KUKA KRL program: EPS_2_251825_SA35_A_20260116064120.src

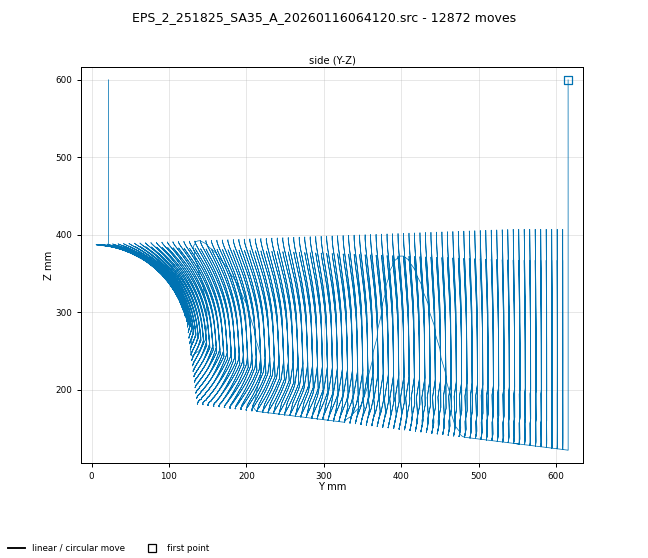
[picture p0: tool path of EPS_2_251825_SA35_A_20260116064120.src, 12872 of 12874 moves have a stored position in this frame; points joined in program order, loops and branches not executed]
&ACCESS RVP
&REL 4
&COMMENT QRS 19112012
&PARAM EDITMASK = *
DEF PART()
EXT BAS (BAS_COMMAND :IN,REAL :IN )
INT I
BAS (#INITMOV,0 )

;KUKA QRS Post kuka4.cps  Date:22-06-2017 !

File_ID=2990

QRS_PRE_INIT()

;Init var - Until changes are made in qrs_pre_init
Outlet_Square_prg=0
Inlet_1_Square_prg=0
Inlet_2_Square_prg=0
Inlet_3_Square_prg=0
Inlet_4_Square_prg=0
Inlet_5_Square_prg=0

Outlet_1={X 0.000, Y 546.330, Z 306.500, B 0.000, E1 0.000 }
Inlet_1={X 0.000, Y 549.180, Z 266.500, B 0.000, E1 180.000 }
Outlet_1_type=201
Inlet_1_type=201
;QRS#1=Sidecore dimensions
;QRS#2=200-8" PVC SDR 35
;QRS#3=200-8" PVC SDR 35
;QRS#4=
;QRS#5=
;QRS#6=
;QRS#7=
;QRS#8=
;QRS#9=12-08 PSX
;QRS#10=12-08 PSX
;QRS#11=
;QRS#12=
;QRS#13=
;QRS#14=
;QRS#15=
;QRS#16=1220x127x686 2,25'
;QRS#17=EPS Height
;QRS#18=407
;QRS#19=*
;QRS#20= UPDATED VERSION 22-06-2017
;QRS#21=*
Outlet_Square=0100
Inlet_1_Square=0100
Inlet_2_Square=0
Inlet_3_Square=0
Inlet_4_Square=0
Inlet_5_Square=0
Mill_Square=1
Outlet_Square_Prg=204
Inlet_1_Square_prg=204

QRS_INIT()

$ADVANCE=5

; T1
PTP {E1 173.649,E2 173.649}
PTP {X 0,Y 615.437,A -85,B 0,C 180,E1 173.649,E2 173.649,E3 0,E4 0,E5 0,E6 0}
QRS_SPEED_INIT()
LIN {X 0,Y 615.437,Z 600,A -85,B 0,C 180,E1 173.649,E2 173.649,E3 0,E4 0,E5 0,E6 0} C_VEL
LIN {X 0,Y 615.437,Z 131.876,A -85,B 0,C 180,E1 173.649,E2 173.649} C_VEL
LIN {X 0,Y 615.437,Z 123.698,A -85,B 0,C 180,E1 173.649,E2 173.649} C_VEL
LIN {X 0,Y 615.425,Z 121.698,A -85,B 0,C 180,E1 173.462,E2 173.462} C_VEL
LIN {X 0,Y 615.423,Z 121.698,A -85,B 0,C 180,E1 171.462,E2 171.462} C_VEL
LIN {X 0,Y 615.422,Z 121.699,A -85,B 0,C 180,E1 169.138,E2 169.138} C_VEL
LIN {X 0,Y 615.448,Z 121.699,A -85,B 0,C 180,E1 166.798,E2 166.798} C_VEL
LIN {X 0,Y 615.463,Z 121.696,A -85,B 0,C 180,E1 164.094,E2 164.094} C_VEL
LIN {X 0,Y 615.423,Z 121.698,A -85,B 0,C 180,E1 161.409,E2 161.409} C_VEL
LIN {X 0,Y 615.498,Z 121.698,A -85,B 0,C 180,E1 158.568,E2 158.568} C_VEL
LIN {X 0,Y 615.427,Z 121.697,A -85,B 0,C 180,E1 155.725,E2 155.725} C_VEL
LIN {X 0,Y 615.428,Z 121.697,A -85,B 0,C 180,E1 153.553,E2 153.553} C_VEL
LIN {X 0,Y 615.483,Z 121.695,A -85,B 0,C 180,E1 150.593,E2 150.593} C_VEL
LIN {X 0,Y 615.452,Z 121.694,A -85,B 0,C 180,E1 148.312,E2 148.312} C_VEL
LIN {X 0,Y 615.431,Z 121.696,A -85,B 0,C 180,E1 145.974,E2 145.974} C_VEL
LIN {X 0,Y 615.487,Z 121.703,A -85,B 0,C 180,E1 143.062,E2 143.062} C_VEL
LIN {X 0,Y 615.436,Z 121.695,A -85,B 0,C 180,E1 140.246,E2 140.246} C_VEL
LIN {X 0,Y 615.434,Z 121.697,A -85,B 0,C 180,E1 137.924,E2 137.924} C_VEL
LIN {X 0,Y 615.442,Z 121.697,A -85,B 0,C 180,E1 135.846,E2 135.846} C_VEL
LIN {X 0,Y 615.488,Z 121.693,A -85,B 0,C 180,E1 133.047,E2 133.047} C_VEL
LIN {X 0,Y 615.448,Z 121.693,A -85,B 0,C 180,E1 130.608,E2 130.608} C_VEL
LIN {X 0,Y 615.447,Z 121.697,A -85,B 0,C 180,E1 128.007,E2 128.007} C_VEL
LIN {X 0,Y 615.489,Z 121.7,A -85,B 0,C 180,E1 125.615,E2 125.615} C_VEL
LIN {X 0,Y 615.486,Z 121.691,A -85,B 0,C 180,E1 123.235,E2 123.235} C_VEL
LIN {X 0,Y 615.457,Z 121.691,A -85,B 0,C 180,E1 120.92,E2 120.92} C_VEL
LIN {X 0,Y 615.441,Z 121.695,A -85,B 0,C 180,E1 118.442,E2 118.442} C_VEL
LIN {X 0,Y 615.493,Z 121.693,A -85,B 0,C 180,E1 115.569,E2 115.569} C_VEL
LIN {X 0,Y 615.446,Z 121.692,A -85,B 0,C 180,E1 112.845,E2 112.845} C_VEL
LIN {X 0,Y 615.449,Z 121.695,A -85,B 0,C 180,E1 110.547,E2 110.547} C_VEL
LIN {X 0,Y 615.45,Z 121.868,A -85,B 0,C 180,E1 108.593,E2 108.593} C_VEL
LIN {X 0,Y 615.493,Z 137.711,A -85,B 0,C 180,E1 105.904,E2 105.904} C_VEL
LIN {X 0,Y 615.469,Z 154.863,A -85,B 0,C 180,E1 103.033,E2 103.033} C_VEL
LIN {X 0,Y 615.476,Z 156.121,A -85,B 0,C 180,E1 102.823,E2 102.823} C_VEL
LIN {X 0,Y 615.483,Z 263.822,A -85,B 0,C 180,E1 101.526,E2 101.526} C_VEL
LIN {X 0,Y 615.474,Z 276.761,A -85,B 0,C 180,E1 101.234,E2 101.234} C_VEL
LIN {X 0,Y 615.487,Z 288.668,A -85,B 0,C 180,E1 100.84,E2 100.84} C_VEL
LIN {X 0,Y 615.481,Z 301.206,A -85,B 0,C 180,E1 100.277,E2 100.277} C_VEL
LIN {X 0,Y 615.494,Z 312.583,A -85,B 0,C 180,E1 99.613,E2 99.613} C_VEL
LIN {X 0,Y 615.498,Z 322.829,A -85,B 0,C 180,E1 98.867,E2 98.867} C_VEL
LIN {X 0,Y 615.498,Z 332.038,A -85,B 0,C 180,E1 98.04,E2 98.04} C_VEL
LIN {X 0,Y 615.499,Z 340.895,A -85,B 0,C 180,E1 97.057,E2 97.057} C_VEL
LIN {X 0,Y 615.497,Z 348.126,A -85,B 0,C 180,E1 96.062,E2 96.062} C_VEL
LIN {X 0,Y 615.497,Z 352.96,A -85,B 0,C 180,E1 95.241,E2 95.241} C_VEL
LIN {X 0,Y 615.494,Z 357.66,A -85,B 0,C 180,E1 94.256,E2 94.256} C_VEL
LIN {X 0,Y 615.494,Z 361.256,A -85,B 0,C 180,E1 93.273,E2 93.273} C_VEL
LIN {X 0,Y 615.496,Z 363.116,A -85,B 0,C 180,E1 92.617,E2 92.617} C_VEL
LIN {X 0,Y 615.5,Z 364.533,A -85,B 0,C 180,E1 91.963,E2 91.963} C_VEL
LIN {X 0,Y 615.496,Z 366.142,A -85,B 0,C 180,E1 90.654,E2 90.654} C_VEL
LIN {X 0,Y 615.495,Z 366.384,A -85,B 0,C 180,E1 90,E2 90} C_VEL
LIN {X 0,Y 615.495,Z 366.205,A -85,B 0,C 180,E1 89.345,E2 89.345} C_VEL
LIN {X 0,Y 615.5,Z 364.682,A -85,B 0,C 180,E1 88.037,E2 88.037} C_VEL
LIN {X 0,Y 615.498,Z 363.341,A -85,B 0,C 180,E1 87.382,E2 87.382} C_VEL
LIN {X 0,Y 615.496,Z 360.493,A -85,B 0,C 180,E1 86.399,E2 86.399} C_VEL
LIN {X 0,Y 615.498,Z 356.633,A -85,B 0,C 180,E1 85.415,E2 85.415} C_VEL
LIN {X 0,Y 615.498,Z 351.65,A -85,B 0,C 180,E1 84.43,E2 84.43} C_VEL
LIN {X 0,Y 615.496,Z 345.208,A -85,B 0,C 180,E1 83.418,E2 83.418} C_VEL
LIN {X 0,Y 615.497,Z 337.535,A -85,B 0,C 180,E1 82.454,E2 82.454} C_VEL
LIN {X 0,Y 615.498,Z 327.756,A -85,B 0,C 180,E1 81.463,E2 81.463} C_VEL
LIN {X 0,Y 615.498,Z 317.49,A -85,B 0,C 180,E1 80.635,E2 80.635} C_VEL
LIN {X 0,Y 615.48,Z 305.928,A -85,B 0,C 180,E1 79.888,E2 79.888} C_VEL
LIN {X 0,Y 615.494,Z 294.071,A -85,B 0,C 180,E1 79.293,E2 79.293} C_VEL
LIN {X 0,Y 615.477,Z 281.156,A -85,B 0,C 180,E1 78.807,E2 78.807} C_VEL
LIN {X 0,Y 615.485,Z 268.552,A -85,B 0,C 180,E1 78.473,E2 78.473} C_VEL
LIN {X 0,Y 615.493,Z 255.419,A -85,B 0,C 180,E1 78.264,E2 78.264} C_VEL
LIN {X 0,Y 615.478,Z 156.153,A -85,B 0,C 180,E1 77.092,E2 77.092} C_VEL
LIN {X 0,Y 615.496,Z 139.253,A -85,B 0,C 180,E1 74.265,E2 74.265} C_VEL
LIN {X 0,Y 615.483,Z 124.248,A -85,B 0,C 180,E1 71.724,E2 71.724} C_VEL
LIN {X 0,Y 615.453,Z 121.694,A -85,B 0,C 180,E1 71.267,E2 71.267} C_VEL
LIN {X 0,Y 615.489,Z 121.686,A -85,B 0,C 180,E1 68.568,E2 68.568} C_VEL
LIN {X 0,Y 615.467,Z 121.697,A -85,B 0,C 180,E1 65.727,E2 65.727} C_VEL
LIN {X 0,Y 615.452,Z 121.695,A -85,B 0,C 180,E1 63.554,E2 63.554} C_VEL
LIN {X 0,Y 615.448,Z 121.692,A -85,B 0,C 180,E1 61.34,E2 61.34} C_VEL
LIN {X 0,Y 615.474,Z 121.688,A -85,B 0,C 180,E1 58.917,E2 58.917} C_VEL
LIN {X 0,Y 615.463,Z 121.697,A -85,B 0,C 180,E1 55.977,E2 55.977} C_VEL
LIN {X 0,Y 615.445,Z 121.693,A -85,B 0,C 180,E1 53.573,E2 53.573} C_VEL
LIN {X 0,Y 615.491,Z 121.688,A -85,B 0,C 180,E1 50.938,E2 50.938} C_VEL
LIN {X 0,Y 615.495,Z 121.701,A -85,B 0,C 180,E1 48.527,E2 48.527} C_VEL
LIN {X 0,Y 615.441,Z 121.694,A -85,B 0,C 180,E1 45.847,E2 45.847} C_VEL
LIN {X 0,Y 615.474,Z 121.69,A -85,B 0,C 180,E1 43.246,E2 43.246} C_VEL
LIN {X 0,Y 615.473,Z 121.7,A -85,B 0,C 180,E1 40.608,E2 40.608} C_VEL
LIN {X 0,Y 615.437,Z 121.696,A -85,B 0,C 180,E1 38.072,E2 38.072} C_VEL
LIN {X 0,Y 615.45,Z 121.693,A -85,B 0,C 180,E1 35.619,E2 35.619} C_VEL
LIN {X 0,Y 615.489,Z 121.694,A -85,B 0,C 180,E1 33.236,E2 33.236} C_VEL
LIN {X 0,Y 615.477,Z 121.701,A -85,B 0,C 180,E1 30.92,E2 30.92} C_VEL
LIN {X 0,Y 615.434,Z 121.697,A -85,B 0,C 180,E1 28.442,E2 28.442} C_VEL
LIN {X 0,Y 615.434,Z 121.697,A -85,B 0,C 180,E1 26.447,E2 26.447} C_VEL
LIN {X 0,Y 615.442,Z 121.694,A -85,B 0,C 180,E1 24,E2 24} C_VEL
LIN {X 0,Y 615.498,Z 121.696,A -85,B 0,C 180,E1 21.432,E2 21.432} C_VEL
LIN {X 0,Y 615.428,Z 121.697,A -85,B 0,C 180,E1 18.59,E2 18.59} C_VEL
LIN {X 0,Y 615.465,Z 121.695,A -85,B 0,C 180,E1 15.906,E2 15.906} C_VEL
LIN {X 0,Y 615.454,Z 121.699,A -85,B 0,C 180,E1 13.202,E2 13.202} C_VEL
LIN {X 0,Y 615.427,Z 121.698,A -85,B 0,C 180,E1 10.861,E2 10.861} C_VEL
LIN {X 0,Y 615.427,Z 121.697,A -85,B 0,C 180,E1 8.538,E2 8.538} C_VEL
LIN {X 0,Y 615.496,Z 121.696,A -85,B 0,C 180,E1 5.899,E2 5.899} C_VEL
LIN {X 0,Y 615.434,Z 121.699,A -85,B 0,C 180,E1 3.273,E2 3.273} C_VEL
LIN {X 0,Y 615.432,Z 121.699,A -85,B 0,C 180,E1 1.309,E2 1.309} C_VEL
LIN {X 0,Y 615.43,Z 121.699,A -85,B 0,C 180,E1 -0.654,E2 -0.654} C_VEL
LIN {X 0,Y 615.428,Z 121.699,A -85,B 0,C 180,E1 -2.618,E2 -2.618} C_VEL
LIN {X 0,Y 615.425,Z 121.7,A -85,B 0,C 180,E1 -4.585,E2 -4.585} C_VEL
LIN {X 0,Y 615.421,Z 121.7,A -85,B 0,C 180,E1 -6.557,E2 -6.557} C_VEL
LIN {X 0,Y 615.421,Z 121.7,A -85,B 0,C 180,E1 -8.538,E2 -8.538} C_VEL
LIN {X 0,Y 615.413,Z 121.7,A -85,B 0,C 180,E1 -10.855,E2 -10.855} C_VEL
LIN {X 0,Y 615.434,Z 121.7,A -85,B 0,C 180,E1 -13.202,E2 -13.202} C_VEL
LIN {X 0,Y 615.461,Z 121.699,A -85,B 0,C 180,E1 -15.906,E2 -15.906} C_VEL
LIN {X 0,Y 615.415,Z 121.7,A -85,B 0,C 180,E1 -18.648,E2 -18.648} C_VEL
LIN {X 0,Y 615.495,Z 121.7,A -85,B 0,C 180,E1 -21.432,E2 -21.432} C_VEL
LIN {X 0,Y 615.419,Z 121.699,A -85,B 0,C 180,E1 -24.275,E2 -24.275} C_VEL
LIN {X 0,Y 615.42,Z 121.699,A -85,B 0,C 180,E1 -26.447,E2 -26.447} C_VEL
LIN {X 0,Y 615.48,Z 121.698,A -85,B 0,C 180,E1 -29.407,E2 -29.407} C_VEL
LIN {X 0,Y 615.449,Z 121.696,A -85,B 0,C 180,E1 -31.688,E2 -31.688} C_VEL
LIN {X 0,Y 615.425,Z 121.697,A -85,B 0,C 180,E1 -34.026,E2 -34.026} C_VEL
LIN {X 0,Y 615.484,Z 121.7,A -85,B 0,C 180,E1 -36.937,E2 -36.937} C_VEL
LIN {X 0,Y 615.499,Z 121.697,A -85,B 0,C 180,E1 -39.064,E2 -39.064} C_VEL
LIN {X 0,Y 615.45,Z 121.695,A -85,B 0,C 180,E1 -41.477,E2 -41.477} C_VEL
LIN {X 0,Y 615.429,Z 121.697,A -85,B 0,C 180,E1 -43.992,E2 -43.992} C_VEL
LIN {X 0,Y 615.429,Z 121.697,A -85,B 0,C 180,E1 -46.008,E2 -46.008} C_VEL
LIN {X 0,Y 615.476,Z 121.699,A -85,B 0,C 180,E1 -48.526,E2 -48.526} C_VEL
LIN {X 0,Y 615.469,Z 121.693,A -85,B 0,C 180,E1 -51.095,E2 -51.095} C_VEL
LIN {X 0,Y 615.434,Z 121.695,A -85,B 0,C 180,E1 -53.572,E2 -53.572} C_VEL
LIN {X 0,Y 615.496,Z 121.701,A -85,B 0,C 180,E1 -56.465,E2 -56.465} C_VEL
LIN {X 0,Y 615.455,Z 121.692,A -85,B 0,C 180,E1 -59.079,E2 -59.079} C_VEL
LIN {X 0,Y 615.438,Z 121.695,A -85,B 0,C 180,E1 -61.559,E2 -61.559} C_VEL
LIN {X 0,Y 615.494,Z 121.695,A -85,B 0,C 180,E1 -64.43,E2 -64.43} C_VEL
LIN {X 0,Y 615.442,Z 121.693,A -85,B 0,C 180,E1 -67.154,E2 -67.154} C_VEL
LIN {X 0,Y 615.441,Z 121.788,A -85,B 0,C 180,E1 -67.44,E2 -67.44} C_VEL
LIN {X 0,Y 615.477,Z 140.398,A -85,B 0,C 180,E1 -69.967,E2 -69.967} C_VEL
LIN {X 0,Y 615.47,Z 161.077,A -85,B 0,C 180,E1 -72.729,E2 -72.729} C_VEL
LIN {X 0,Y 615.472,Z 181.732,A -85,B 0,C 180,E1 -75.45,E2 -75.45} C_VEL
LIN {X 0,Y 615.454,Z 194.469,A -85,B 0,C 180,E1 -77.113,E2 -77.113} C_VEL
LIN {X 0,Y 615.488,Z 302.82,A -85,B 0,C 180,E1 -78.41,E2 -78.41} C_VEL
LIN {X 0,Y 615.477,Z 315.339,A -85,B 0,C 180,E1 -78.681,E2 -78.681} C_VEL
LIN {X 0,Y 615.488,Z 328.617,A -85,B 0,C 180,E1 -79.113,E2 -79.113} C_VEL
LIN {X 0,Y 615.477,Z 340.475,A -85,B 0,C 180,E1 -79.639,E2 -79.639} C_VEL
LIN {X 0,Y 615.494,Z 351.991,A -85,B 0,C 180,E1 -80.304,E2 -80.304} C_VEL
LIN {X 0,Y 615.499,Z 362.338,A -85,B 0,C 180,E1 -81.05,E2 -81.05} C_VEL
LIN {X 0,Y 615.497,Z 370.809,A -85,B 0,C 180,E1 -81.794,E2 -81.794} C_VEL
LIN {X 0,Y 615.498,Z 378.604,A -85,B 0,C 180,E1 -82.619,E2 -82.619} C_VEL
LIN {X 0,Y 615.496,Z 386.201,A -85,B 0,C 180,E1 -83.608,E2 -83.608} C_VEL
LIN {X 0,Y 615.498,Z 393.203,A -85,B 0,C 180,E1 -84.759,E2 -84.759} C_VEL
LIN {X 0,Y 615.494,Z 397.85,A -85,B 0,C 180,E1 -85.743,E2 -85.743} C_VEL
LIN {X 0,Y 615.494,Z 401.398,A -85,B 0,C 180,E1 -86.727,E2 -86.727} C_VEL
LIN {X 0,Y 615.497,Z 403.232,A -85,B 0,C 180,E1 -87.382,E2 -87.382} C_VEL
LIN {X 0,Y 615.5,Z 404.607,A -85,B 0,C 180,E1 -88.037,E2 -88.037} C_VEL
LIN {X 0,Y 615.496,Z 406.173,A -85,B 0,C 180,E1 -89.345,E2 -89.345} C_VEL
LIN {X 0,Y 615.494,Z 406.389,A -85,B 0,C 180,E1 -90,E2 -90} C_VEL
LIN {X 0,Y 615.495,Z 405.58,A -85,B 0,C 180,E1 -91.308,E2 -91.308} C_VEL
LIN {X 0,Y 615.5,Z 404.608,A -85,B 0,C 180,E1 -91.963,E2 -91.963} C_VEL
LIN {X 0,Y 615.497,Z 403.234,A -85,B 0,C 180,E1 -92.617,E2 -92.617} C_VEL
LIN {X 0,Y 615.496,Z 400.351,A -85,B 0,C 180,E1 -93.6,E2 -93.6} C_VEL
LIN {X 0,Y 615.498,Z 396.443,A -85,B 0,C 180,E1 -94.584,E2 -94.584} C_VEL
LIN {X 0,Y 615.499,Z 391.407,A -85,B 0,C 180,E1 -95.569,E2 -95.569} C_VEL
LIN {X 0,Y 615.497,Z 384.869,A -85,B 0,C 180,E1 -96.583,E2 -96.583} C_VEL
LIN {X 0,Y 615.497,Z 377.137,A -85,B 0,C 180,E1 -97.545,E2 -97.545} C_VEL
LIN {X 0,Y 615.498,Z 369.05,A -85,B 0,C 180,E1 -98.371,E2 -98.371} C_VEL
LIN {X 0,Y 615.499,Z 359.174,A -85,B 0,C 180,E1 -99.198,E2 -99.198} C_VEL
LIN {X 0,Y 615.488,Z 347.99,A -85,B 0,C 180,E1 -99.945,E2 -99.945} C_VEL
LIN {X 0,Y 615.482,Z 337.034,A -85,B 0,C 180,E1 -100.527,E2 -100.527} C_VEL
LIN {X 0,Y 615.48,Z 324.497,A -85,B 0,C 180,E1 -101.04,E2 -101.04} C_VEL
LIN {X 0,Y 615.479,Z 312.09,A -85,B 0,C 180,E1 -101.401,E2 -101.401} C_VEL
LIN {X 0,Y 615.493,Z 298.502,A -85,B 0,C 180,E1 -101.651,E2 -101.651} C_VEL
LIN {X 0,Y 615.454,Z 194.475,A -85,B 0,C 180,E1 -102.887,E2 -102.887} C_VEL
LIN {X 0,Y 615.496,Z 172.701,A -85,B 0,C 180,E1 -105.734,E2 -105.734} C_VEL
LIN {X 0,Y 615.455,Z 152.32,A -85,B 0,C 180,E1 -108.436,E2 -108.436} C_VEL
LIN {X 0,Y 615.475,Z 132.642,A -85,B 0,C 180,E1 -111.081,E2 -111.081} C_VEL
LIN {X 0,Y 615.44,Z 121.695,A -85,B 0,C 180,E1 -112.591,E2 -112.591} C_VEL
LIN {X 0,Y 615.452,Z 121.692,A -85,B 0,C 180,E1 -114.993,E2 -114.993} C_VEL
LIN {X 0,Y 615.472,Z 121.699,A -85,B 0,C 180,E1 -117.915,E2 -117.915} C_VEL
LIN {X 0,Y 615.446,Z 121.697,A -85,B 0,C 180,E1 -120.161,E2 -120.161} C_VEL
LIN {X 0,Y 615.436,Z 121.695,A -85,B 0,C 180,E1 -122.46,E2 -122.46} C_VEL
LIN {X 0,Y 615.453,Z 121.693,A -85,B 0,C 180,E1 -124.816,E2 -124.816} C_VEL
LIN {X 0,Y 615.498,Z 121.694,A -85,B 0,C 180,E1 -127.24,E2 -127.24} C_VEL
LIN {X 0,Y 615.454,Z 121.698,A -85,B 0,C 180,E1 -129.752,E2 -129.752} C_VEL
LIN {X 0,Y 615.431,Z 121.697,A -85,B 0,C 180,E1 -132.074,E2 -132.074} C_VEL
LIN {X 0,Y 615.43,Z 121.696,A -85,B 0,C 180,E1 -134.153,E2 -134.153} C_VEL
LIN {X 0,Y 615.471,Z 121.693,A -85,B 0,C 180,E1 -136.754,E2 -136.754} C_VEL
LIN {X 0,Y 615.457,Z 121.7,A -85,B 0,C 180,E1 -139.391,E2 -139.391} C_VEL
LIN {X 0,Y 615.493,Z 121.7,A -85,B 0,C 180,E1 -141.096,E2 -141.096} C_VEL
LIN {X 0,Y 615.432,Z 121.699,A -85,B 0,C 180,E1 -143.571,E2 -143.571} C_VEL
LIN {X 0,Y 615.427,Z 121.697,A -85,B 0,C 180,E1 -145.974,E2 -145.974} C_VEL
LIN {X 0,Y 615.482,Z 121.701,A -85,B 0,C 180,E1 -148.913,E2 -148.913} C_VEL
LIN {X 0,Y 615.424,Z 121.698,A -85,B 0,C 180,E1 -151.558,E2 -151.558} C_VEL
LIN {X 0,Y 615.422,Z 121.698,A -85,B 0,C 180,E1 -153.553,E2 -153.553} C_VEL
LIN {X 0,Y 615.436,Z 121.697,A -85,B 0,C 180,E1 -156,E2 -156} C_VEL
LIN {X 0,Y 615.498,Z 121.7,A -85,B 0,C 180,E1 -158.568,E2 -158.568} C_VEL
LIN {X 0,Y 615.415,Z 121.7,A -85,B 0,C 180,E1 -161.412,E2 -161.412} C_VEL
LIN {X 0,Y 615.462,Z 121.698,A -85,B 0,C 180,E1 -164.094,E2 -164.094} C_VEL
LIN {X 0,Y 615.439,Z 121.7,A -85,B 0,C 180,E1 -166.798,E2 -166.798} C_VEL
LIN {X 0,Y 615.415,Z 121.7,A -85,B 0,C 180,E1 -169.141,E2 -169.141} C_VEL
LIN {X 0,Y 615.419,Z 121.7,A -85,B 0,C 180,E1 -171.462,E2 -171.462} C_VEL
LIN {X 0,Y 615.496,Z 121.7,A -85,B 0,C 180,E1 -174.102,E2 -174.102} C_VEL
LIN {X 0,Y 615.422,Z 121.7,A -85,B 0,C 180,E1 -176.727,E2 -176.727} C_VEL
LIN {X 0,Y 615.422,Z 121.7,A -85,B 0,C 180,E1 -178.691,E2 -178.691} C_VEL
LIN {X 0,Y 615.423,Z 121.699,A -85,B 0,C 180,E1 -180.654,E2 -180.654} C_VEL
LIN {X 0,Y 615.424,Z 121.699,A -85,B 0,C 180,E1 -182.618,E2 -182.618} C_VEL
LIN {X 0,Y 615.424,Z 121.699,A -85,B 0,C 180,E1 -184.585,E2 -184.585} C_VEL
LIN {X 0,Y 615.425,Z 121.698,A -85,B 0,C 180,E1 -186.538,E2 -186.538} C_VEL
LIN {X 0,Y 614.752,Z 121.846,A -85,B 0,C 180,E1 -187.084,E2 -187.084} C_VEL
LIN {X 0,Y 611.92,Z 122.262,A -85,B 0,C 180,E1 -187.97,E2 -187.97} C_VEL
LIN {X 0,Y 609.535,Z 122.57,A -85,B 0,C 180,E1 -188.683,E2 -188.683} C_VEL
LIN {X 0,Y 608.512,Z 122.685,A -85,B 0,C 180,E1 -189.233,E2 -189.233} C_VEL
LIN {X 0,Y 608.428,Z 122.694,A -85,B 0,C 180,E1 -189.419,E2 -189.419} C_VEL
LIN {X 0,Y 608.441,Z 122.693,A -85,B 0,C 180,E1 -192,E2 -192} C_VEL
LIN {X 0,Y 608.394,Z 122.695,A -85,B 0,C 180,E1 -194.723,E2 -194.723} C_VEL
LIN {X 0,Y 608.431,Z 122.701,A -85,B 0,C 180,E1 -197.477,E2 -197.477} C_VEL
LIN {X 0,Y 608.413,Z 122.693,A -85,B 0,C 180,E1 -200.276,E2 -200.276} C_VEL
LIN {X 0,Y 608.419,Z 122.692,A -85,B 0,C 180,E1 -202.47,E2 -202.47} C_VEL
LIN {X 0,Y 608.436,Z 122.7,A -85,B 0,C 180,E1 -205.302,E2 -205.302} C_VEL
LIN {X 0,Y 608.429,Z 122.696,A -85,B 0,C 180,E1 -207.519,E2 -207.519} C_VEL
LIN {X 0,Y 608.408,Z 122.693,A -85,B 0,C 180,E1 -209.964,E2 -209.964} C_VEL
LIN {X 0,Y 608.42,Z 122.694,A -85,B 0,C 180,E1 -212.518,E2 -212.518} C_VEL
LIN {X 0,Y 608.419,Z 122.697,A -85,B 0,C 180,E1 -215.279,E2 -215.279} C_VEL
LIN {X 0,Y 608.435,Z 122.69,A -85,B 0,C 180,E1 -217.749,E2 -217.749} C_VEL
LIN {X 0,Y 608.426,Z 122.693,A -85,B 0,C 180,E1 -220.328,E2 -220.328} C_VEL
LIN {X 0,Y 608.46,Z 122.689,A -85,B 0,C 180,E1 -223.309,E2 -223.309} C_VEL
LIN {X 0,Y 608.434,Z 122.692,A -85,B 0,C 180,E1 -226.129,E2 -226.129} C_VEL
LIN {X 0,Y 608.457,Z 122.694,A -85,B 0,C 180,E1 -228.825,E2 -228.825} C_VEL
LIN {X 0,Y 608.435,Z 122.69,A -85,B 0,C 180,E1 -231.764,E2 -231.764} C_VEL
LIN {X 0,Y 608.433,Z 122.693,A -85,B 0,C 180,E1 -233.957,E2 -233.957} C_VEL
LIN {X 0,Y 608.464,Z 122.696,A -85,B 0,C 180,E1 -236.33,E2 -236.33} C_VEL
LIN {X 0,Y 608.443,Z 122.693,A -85,B 0,C 180,E1 -238.734,E2 -238.734} C_VEL
LIN {X 0,Y 608.435,Z 122.69,A -85,B 0,C 180,E1 -241.387,E2 -241.387} C_VEL
LIN {X 0,Y 608.433,Z 122.697,A -85,B 0,C 180,E1 -243.965,E2 -243.965} C_VEL
LIN {X 0,Y 608.432,Z 122.691,A -85,B 0,C 180,E1 -246.876,E2 -246.876} C_VEL
LIN {X 0,Y 608.438,Z 122.691,A -85,B 0,C 180,E1 -249.33,E2 -249.33} C_VEL
LIN {X 0,Y 608.462,Z 122.864,A -85,B 0,C 180,E1 -251.345,E2 -251.345} C_VEL
LIN {X 0,Y 608.499,Z 138.846,A -85,B 0,C 180,E1 -254.08,E2 -254.08} C_VEL
LIN {X 0,Y 608.448,Z 155.056,A -85,B 0,C 180,E1 -256.814,E2 -256.814} C_VEL
LIN {X 0,Y 608.464,Z 156.323,A -85,B 0,C 180,E1 -257.026,E2 -257.026} C_VEL
LIN {X 0,Y 608.56,Z 165.703,A -85,B 0,C 180,E1 -257.156,E2 -257.156} C_VEL
LIN {X 0,Y 608.554,Z 262.824,A -85,B 0,C 180,E1 -258.32,E2 -258.32} C_VEL
LIN {X 0,Y 608.524,Z 276.133,A -85,B 0,C 180,E1 -258.614,E2 -258.614} C_VEL
LIN {X 0,Y 608.522,Z 289.437,A -85,B 0,C 180,E1 -259.058,E2 -259.058} C_VEL
LIN {X 0,Y 608.494,Z 301.378,A -85,B 0,C 180,E1 -259.604,E2 -259.604} C_VEL
LIN {X 0,Y 608.506,Z 312.797,A -85,B 0,C 180,E1 -260.276,E2 -260.276} C_VEL
LIN {X 0,Y 608.474,Z 323.09,A -85,B 0,C 180,E1 -261.03,E2 -261.03} C_VEL
LIN {X 0,Y 608.464,Z 332.354,A -85,B 0,C 180,E1 -261.866,E2 -261.866} C_VEL
LIN {X 0,Y 608.466,Z 341.327,A -85,B 0,C 180,E1 -262.868,E2 -262.868} C_VEL
LIN {X 0,Y 608.444,Z 348.558,A -85,B 0,C 180,E1 -263.867,E2 -263.867} C_VEL
LIN {X 0,Y 608.462,Z 353.437,A -85,B 0,C 180,E1 -264.699,E2 -264.699} C_VEL
LIN {X 0,Y 608.439,Z 358.18,A -85,B 0,C 180,E1 -265.695,E2 -265.695} C_VEL
LIN {X 0,Y 608.425,Z 361.813,A -85,B 0,C 180,E1 -266.689,E2 -266.689} C_VEL
LIN {X 0,Y 608.425,Z 363.692,A -85,B 0,C 180,E1 -267.352,E2 -267.352} C_VEL
LIN {X 0,Y 608.445,Z 365.127,A -85,B 0,C 180,E1 -268.015,E2 -268.015} C_VEL
LIN {X 0,Y 608.439,Z 366.752,A -85,B 0,C 180,E1 -269.339,E2 -269.339} C_VEL
LIN {X 0,Y 608.435,Z 366.996,A -85,B 0,C 180,E1 -270,E2 -270} C_VEL
LIN {X 0,Y 608.438,Z 366.815,A -85,B 0,C 180,E1 -270.662,E2 -270.662} C_VEL
LIN {X 0,Y 608.445,Z 365.276,A -85,B 0,C 180,E1 -271.986,E2 -271.986} C_VEL
LIN {X 0,Y 608.426,Z 363.918,A -85,B 0,C 180,E1 -272.649,E2 -272.649} C_VEL
LIN {X 0,Y 608.449,Z 361.041,A -85,B 0,C 180,E1 -273.643,E2 -273.643} C_VEL
LIN {X 0,Y 608.433,Z 357.142,A -85,B 0,C 180,E1 -274.638,E2 -274.638} C_VEL
LIN {X 0,Y 608.45,Z 352.111,A -85,B 0,C 180,E1 -275.635,E2 -275.635} C_VEL
LIN {X 0,Y 608.441,Z 345.793,A -85,B 0,C 180,E1 -276.633,E2 -276.633} C_VEL
LIN {X 0,Y 608.475,Z 337.876,A -85,B 0,C 180,E1 -277.633,E2 -277.633} C_VEL
LIN {X 0,Y 608.472,Z 328.034,A -85,B 0,C 180,E1 -278.636,E2 -278.636} C_VEL
LIN {X 0,Y 608.48,Z 317.711,A -85,B 0,C 180,E1 -279.474,E2 -279.474} C_VEL
LIN {X 0,Y 608.476,Z 306.096,A -85,B 0,C 180,E1 -280.229,E2 -280.229} C_VEL
LIN {X 0,Y 608.51,Z 294.204,A -85,B 0,C 180,E1 -280.831,E2 -280.831} C_VEL
LIN {X 0,Y 608.52,Z 281.256,A -85,B 0,C 180,E1 -281.323,E2 -281.323} C_VEL
LIN {X 0,Y 608.544,Z 268.637,A -85,B 0,C 180,E1 -281.66,E2 -281.66} C_VEL
LIN {X 0,Y 608.556,Z 255.527,A -85,B 0,C 180,E1 -281.871,E2 -281.871} C_VEL
LIN {X 0,Y 608.45,Z 156.349,A -85,B 0,C 180,E1 -283.059,E2 -283.059} C_VEL
LIN {X 0,Y 608.497,Z 139.372,A -85,B 0,C 180,E1 -285.921,E2 -285.921} C_VEL
LIN {X 0,Y 608.47,Z 122.894,A -85,B 0,C 180,E1 -288.739,E2 -288.739} C_VEL
LIN {X 0,Y 608.441,Z 122.689,A -85,B 0,C 180,E1 -290.982,E2 -290.982} C_VEL
LIN {X 0,Y 608.469,Z 122.694,A -85,B 0,C 180,E1 -293.845,E2 -293.845} C_VEL
LIN {X 0,Y 608.436,Z 122.698,A -85,B 0,C 180,E1 -296.036,E2 -296.036} C_VEL
LIN {X 0,Y 608.442,Z 122.689,A -85,B 0,C 180,E1 -298.614,E2 -298.614} C_VEL
LIN {X 0,Y 608.446,Z 122.691,A -85,B 0,C 180,E1 -301.267,E2 -301.267} C_VEL
LIN {X 0,Y 608.474,Z 122.695,A -85,B 0,C 180,E1 -303.735,E2 -303.735} C_VEL
LIN {X 0,Y 608.437,Z 122.692,A -85,B 0,C 180,E1 -306.093,E2 -306.093} C_VEL
LIN {X 0,Y 608.421,Z 122.692,A -85,B 0,C 180,E1 -308.591,E2 -308.591} C_VEL
LIN {X 0,Y 608.468,Z 122.694,A -85,B 0,C 180,E1 -311.342,E2 -311.342} C_VEL
LIN {X 0,Y 608.44,Z 122.692,A -85,B 0,C 180,E1 -313.872,E2 -313.872} C_VEL
LIN {X 0,Y 608.462,Z 122.688,A -85,B 0,C 180,E1 -316.692,E2 -316.692} C_VEL
LIN {X 0,Y 608.431,Z 122.694,A -85,B 0,C 180,E1 -319.673,E2 -319.673} C_VEL
LIN {X 0,Y 608.439,Z 122.689,A -85,B 0,C 180,E1 -322.251,E2 -322.251} C_VEL
LIN {X 0,Y 608.445,Z 122.699,A -85,B 0,C 180,E1 -325.095,E2 -325.095} C_VEL
LIN {X 0,Y 608.426,Z 122.691,A -85,B 0,C 180,E1 -327.903,E2 -327.903} C_VEL
LIN {X 0,Y 608.435,Z 122.691,A -85,B 0,C 180,E1 -330.219,E2 -330.219} C_VEL
LIN {X 0,Y 608.481,Z 122.694,A -85,B 0,C 180,E1 -332.791,E2 -332.791} C_VEL
LIN {X 0,Y 608.421,Z 122.693,A -85,B 0,C 180,E1 -335.427,E2 -335.427} C_VEL
LIN {X 0,Y 608.457,Z 122.691,A -85,B 0,C 180,E1 -338.308,E2 -338.308} C_VEL
LIN {X 0,Y 608.413,Z 122.694,A -85,B 0,C 180,E1 -341.299,E2 -341.299} C_VEL
LIN {X 0,Y 608.427,Z 122.692,A -85,B 0,C 180,E1 -343.905,E2 -343.905} C_VEL
LIN {X 0,Y 608.438,Z 122.697,A -85,B 0,C 180,E1 -346.643,E2 -346.643} C_VEL
LIN {X 0,Y 608.408,Z 122.693,A -85,B 0,C 180,E1 -349.349,E2 -349.349} C_VEL
LIN {X 0,Y 608.467,Z 122.692,A -85,B 0,C 180,E1 -352.033,E2 -352.033} C_VEL
LIN {X 0,Y 608.424,Z 122.694,A -85,B 0,C 180,E1 -354.698,E2 -354.698} C_VEL
LIN {X 0,Y 608.422,Z 122.692,A -85,B 0,C 180,E1 -357.352,E2 -357.352} C_VEL
LIN {X 0,Y 608.471,Z 122.695,A -85,B 0,C 180,E1 -360,E2 -360} C_VEL
LIN {X 0,Y 608.424,Z 122.693,A -85,B 0,C 180,E1 -362.648,E2 -362.648} C_VEL
LIN {X 0,Y 608.412,Z 122.694,A -85,B 0,C 180,E1 -365.302,E2 -365.302} C_VEL
LIN {X 0,Y 608.461,Z 122.695,A -85,B 0,C 180,E1 -367.967,E2 -367.967} C_VEL
LIN {X 0,Y 608.398,Z 122.695,A -85,B 0,C 180,E1 -370.651,E2 -370.651} C_VEL
LIN {X 0,Y 608.423,Z 122.696,A -85,B 0,C 180,E1 -373.357,E2 -373.357} C_VEL
LIN {X 0,Y 608.421,Z 122.695,A -85,B 0,C 180,E1 -376.095,E2 -376.095} C_VEL
LIN {X 0,Y 608.422,Z 122.693,A -85,B 0,C 180,E1 -378.871,E2 -378.871} C_VEL
LIN {X 0,Y 608.452,Z 122.694,A -85,B 0,C 180,E1 -381.692,E2 -381.692} C_VEL
LIN {X 0,Y 608.406,Z 122.694,A -85,B 0,C 180,E1 -384.573,E2 -384.573} C_VEL
LIN {X 0,Y 608.467,Z 122.695,A -85,B 0,C 180,E1 -387.206,E2 -387.206} C_VEL
LIN {X 0,Y 608.404,Z 122.694,A -85,B 0,C 180,E1 -389.962,E2 -389.962} C_VEL
LIN {X 0,Y 608.413,Z 122.694,A -85,B 0,C 180,E1 -392.516,E2 -392.516} C_VEL
LIN {X 0,Y 608.413,Z 122.699,A -85,B 0,C 180,E1 -395.28,E2 -395.28} C_VEL
LIN {X 0,Y 608.431,Z 122.691,A -85,B 0,C 180,E1 -397.749,E2 -397.749} C_VEL
LIN {X 0,Y 608.431,Z 122.692,A -85,B 0,C 180,E1 -400.327,E2 -400.327} C_VEL
LIN {X 0,Y 608.459,Z 122.69,A -85,B 0,C 180,E1 -403.308,E2 -403.308} C_VEL
LIN {X 0,Y 608.427,Z 122.692,A -85,B 0,C 180,E1 -406.127,E2 -406.127} C_VEL
LIN {X 0,Y 608.455,Z 122.695,A -85,B 0,C 180,E1 -408.824,E2 -408.824} C_VEL
LIN {X 0,Y 608.412,Z 122.693,A -85,B 0,C 180,E1 -411.408,E2 -411.408} C_VEL
LIN {X 0,Y 608.43,Z 122.692,A -85,B 0,C 180,E1 -413.907,E2 -413.907} C_VEL
LIN {X 0,Y 608.447,Z 122.696,A -85,B 0,C 180,E1 -416.328,E2 -416.328} C_VEL
LIN {X 0,Y 608.444,Z 122.694,A -85,B 0,C 180,E1 -418.733,E2 -418.733} C_VEL
LIN {X 0,Y 608.433,Z 122.69,A -85,B 0,C 180,E1 -421.387,E2 -421.387} C_VEL
LIN {X 0,Y 608.43,Z 122.696,A -85,B 0,C 180,E1 -423.964,E2 -423.964} C_VEL
LIN {X 0,Y 608.43,Z 122.693,A -85,B 0,C 180,E1 -426.875,E2 -426.875} C_VEL
LIN {X 0,Y 608.435,Z 122.82,A -85,B 0,C 180,E1 -427.309,E2 -427.309} C_VEL
LIN {X 0,Y 608.573,Z 138.08,A -85,B 0,C 180,E1 -429.412,E2 -429.412} C_VEL
LIN {X 0,Y 608.532,Z 158.529,A -85,B 0,C 180,E1 -432.179,E2 -432.179} C_VEL
LIN {X 0,Y 608.493,Z 179.24,A -85,B 0,C 180,E1 -434.937,E2 -434.937} C_VEL
LIN {X 0,Y 608.441,Z 194.612,A -85,B 0,C 180,E1 -436.962,E2 -436.962} C_VEL
LIN {X 0,Y 608.564,Z 247,A -85,B 0,C 180,E1 -437.6,E2 -437.6} C_VEL
LIN {X 0,Y 608.547,Z 302.937,A -85,B 0,C 180,E1 -438.276,E2 -438.276} C_VEL
LIN {X 0,Y 608.512,Z 316.21,A -85,B 0,C 180,E1 -438.571,E2 -438.571} C_VEL
LIN {X 0,Y 608.514,Z 328.627,A -85,B 0,C 180,E1 -438.982,E2 -438.982} C_VEL
LIN {X 0,Y 608.499,Z 340.631,A -85,B 0,C 180,E1 -439.519,E2 -439.519} C_VEL
LIN {X 0,Y 608.484,Z 352.194,A -85,B 0,C 180,E1 -440.191,E2 -440.191} C_VEL
LIN {X 0,Y 608.485,Z 362.591,A -85,B 0,C 180,E1 -440.946,E2 -440.946} C_VEL
LIN {X 0,Y 608.475,Z 371.109,A -85,B 0,C 180,E1 -441.699,E2 -441.699} C_VEL
LIN {X 0,Y 608.471,Z 378.958,A -85,B 0,C 180,E1 -442.534,E2 -442.534} C_VEL
LIN {X 0,Y 608.461,Z 386.286,A -85,B 0,C 180,E1 -443.484,E2 -443.484} C_VEL
LIN {X 0,Y 608.451,Z 391.864,A -85,B 0,C 180,E1 -444.365,E2 -444.365} C_VEL
LIN {X 0,Y 608.432,Z 396.949,A -85,B 0,C 180,E1 -445.362,E2 -445.362} C_VEL
LIN {X 0,Y 608.449,Z 400.895,A -85,B 0,C 180,E1 -446.357,E2 -446.357} C_VEL
LIN {X 0,Y 608.425,Z 403.808,A -85,B 0,C 180,E1 -447.351,E2 -447.351} C_VEL
LIN {X 0,Y 608.445,Z 405.201,A -85,B 0,C 180,E1 -448.014,E2 -448.014} C_VEL
LIN {X 0,Y 608.438,Z 406.783,A -85,B 0,C 180,E1 -449.338,E2 -449.338} C_VEL
LIN {X 0,Y 608.434,Z 407,A -85,B 0,C 180,E1 -450,E2 -450} C_VEL
LIN {X 0,Y 608.448,Z 406.184,A -85,B 0,C 180,E1 -451.323,E2 -451.323} C_VEL
LIN {X 0,Y 608.445,Z 405.202,A -85,B 0,C 180,E1 -451.985,E2 -451.985} C_VEL
LIN {X 0,Y 608.425,Z 403.81,A -85,B 0,C 180,E1 -452.648,E2 -452.648} C_VEL
LIN {X 0,Y 608.449,Z 400.897,A -85,B 0,C 180,E1 -453.642,E2 -453.642} C_VEL
LIN {X 0,Y 608.432,Z 396.952,A -85,B 0,C 180,E1 -454.637,E2 -454.637} C_VEL
LIN {X 0,Y 608.438,Z 390.879,A -85,B 0,C 180,E1 -455.8,E2 -455.8} C_VEL
LIN {X 0,Y 608.462,Z 384.238,A -85,B 0,C 180,E1 -456.799,E2 -456.799} C_VEL
LIN {X 0,Y 608.456,Z 375.993,A -85,B 0,C 180,E1 -457.8,E2 -457.8} C_VEL
LIN {X 0,Y 608.472,Z 367.542,A -85,B 0,C 180,E1 -458.635,E2 -458.635} C_VEL
LIN {X 0,Y 608.479,Z 357.098,A -85,B 0,C 180,E1 -459.473,E2 -459.473} C_VEL
LIN {X 0,Y 608.489,Z 346.764,A -85,B 0,C 180,E1 -460.144,E2 -460.144} C_VEL
LIN {X 0,Y 608.519,Z 335.275,A -85,B 0,C 180,E1 -460.74,E2 -460.74} C_VEL
LIN {X 0,Y 608.528,Z 322.903,A -85,B 0,C 180,E1 -461.224,E2 -461.224} C_VEL
LIN {X 0,Y 608.544,Z 309.461,A -85,B 0,C 180,E1 -461.596,E2 -461.596} C_VEL
LIN {X 0,Y 608.553,Z 297.125,A -85,B 0,C 180,E1 -461.807,E2 -461.807} C_VEL
LIN {X 0,Y 608.496,Z 195.189,A -85,B 0,C 180,E1 -463.015,E2 -463.015} C_VEL
LIN {X 0,Y 608.444,Z 194.132,A -85,B 0,C 180,E1 -463.101,E2 -463.101} C_VEL
LIN {X 0,Y 608.497,Z 172.773,A -85,B 0,C 180,E1 -465.92,E2 -465.92} C_VEL
LIN {X 0,Y 608.498,Z 151.84,A -85,B 0,C 180,E1 -468.723,E2 -468.723} C_VEL
LIN {X 0,Y 608.574,Z 131.351,A -85,B 0,C 180,E1 -471.509,E2 -471.509} C_VEL
LIN {X 0,Y 608.424,Z 122.693,A -85,B 0,C 180,E1 -472.715,E2 -472.715} C_VEL
LIN {X 0,Y 608.438,Z 122.693,A -85,B 0,C 180,E1 -475.301,E2 -475.301} C_VEL
LIN {X 0,Y 608.437,Z 122.697,A -85,B 0,C 180,E1 -477.518,E2 -477.518} C_VEL
LIN {X 0,Y 608.433,Z 122.695,A -85,B 0,C 180,E1 -479.965,E2 -479.965} C_VEL
LIN {X 0,Y 608.419,Z 122.692,A -85,B 0,C 180,E1 -482.516,E2 -482.516} C_VEL
LIN {X 0,Y 608.422,Z 122.693,A -85,B 0,C 180,E1 -484.901,E2 -484.901} C_VEL
LIN {X 0,Y 608.442,Z 122.694,A -85,B 0,C 180,E1 -487.747,E2 -487.747} C_VEL
LIN {X 0,Y 608.427,Z 122.691,A -85,B 0,C 180,E1 -490.326,E2 -490.326} C_VEL
LIN {X 0,Y 608.481,Z 122.694,A -85,B 0,C 180,E1 -493.31,E2 -493.31} C_VEL
LIN {X 0,Y 608.425,Z 122.691,A -85,B 0,C 180,E1 -496.126,E2 -496.126} C_VEL
LIN {X 0,Y 608.448,Z 122.694,A -85,B 0,C 180,E1 -498.823,E2 -498.823} C_VEL
LIN {X 0,Y 608.424,Z 122.692,A -85,B 0,C 180,E1 -501.763,E2 -501.763} C_VEL
LIN {X 0,Y 608.42,Z 122.692,A -85,B 0,C 180,E1 -503.956,E2 -503.956} C_VEL
LIN {X 0,Y 608.434,Z 122.692,A -85,B 0,C 180,E1 -506.327,E2 -506.327} C_VEL
LIN {X 0,Y 608.438,Z 122.698,A -85,B 0,C 180,E1 -508.732,E2 -508.732} C_VEL
LIN {X 0,Y 608.424,Z 122.693,A -85,B 0,C 180,E1 -511.386,E2 -511.386} C_VEL
LIN {X 0,Y 608.409,Z 122.696,A -85,B 0,C 180,E1 -513.224,E2 -513.224} C_VEL
LIN {X 0,Y 608.407,Z 122.694,A -85,B 0,C 180,E1 -515.86,E2 -515.86} C_VEL
LIN {X 0,Y 608.454,Z 122.693,A -85,B 0,C 180,E1 -518.308,E2 -518.308} C_VEL
LIN {X 0,Y 608.402,Z 122.694,A -85,B 0,C 180,E1 -521.3,E2 -521.3} C_VEL
LIN {X 0,Y 608.422,Z 122.694,A -85,B 0,C 180,E1 -523.905,E2 -523.905} C_VEL
LIN {X 0,Y 608.426,Z 122.696,A -85,B 0,C 180,E1 -526.643,E2 -526.643} C_VEL
LIN {X 0,Y 608.399,Z 122.694,A -85,B 0,C 180,E1 -529.349,E2 -529.349} C_VEL
LIN {X 0,Y 608.458,Z 122.695,A -85,B 0,C 180,E1 -532.033,E2 -532.033} C_VEL
LIN {X 0,Y 608.412,Z 122.695,A -85,B 0,C 180,E1 -534.698,E2 -534.698} C_VEL
LIN {X 0,Y 608.416,Z 122.693,A -85,B 0,C 180,E1 -537.352,E2 -537.352} C_VEL
LIN {X 0,Y 608.466,Z 122.696,A -85,B 0,C 180,E1 -540,E2 -540} C_VEL
LIN {X 0,Y 608.419,Z 122.692,A -85,B 0,C 180,E1 -542.648,E2 -542.648} C_VEL
LIN {X 0,Y 608.418,Z 122.694,A -85,B 0,C 180,E1 -545.302,E2 -545.302} C_VEL
LIN {X 0,Y 608.463,Z 122.693,A -85,B 0,C 180,E1 -547.967,E2 -547.967} C_VEL
LIN {X 0,Y 608.428,Z 122.694,A -85,B 0,C 180,E1 -549.419,E2 -549.419} C_VEL
LIN {X 0,Y 607.765,Z 122.779,A -85,B 0,C 180,E1 -549.971,E2 -549.971} C_VEL
LIN {X 0,Y 604.926,Z 123.131,A -85,B 0,C 180,E1 -550.868,E2 -550.868} C_VEL
LIN {X 0,Y 602.515,Z 123.437,A -85,B 0,C 180,E1 -551.589,E2 -551.589} C_VEL
LIN {X 0,Y 601.463,Z 123.561,A -85,B 0,C 180,E1 -552.146,E2 -552.146} C_VEL
LIN {X 0,Y 601.369,Z 123.571,A -85,B 0,C 180,E1 -552.334,E2 -552.334} C_VEL
LIN {X 0,Y 601.371,Z 123.571,A -85,B 0,C 180,E1 -554.899,E2 -554.899} C_VEL
LIN {X 0,Y 601.37,Z 123.577,A -85,B 0,C 180,E1 -557.689,E2 -557.689} C_VEL
LIN {X 0,Y 601.378,Z 123.573,A -85,B 0,C 180,E1 -559.81,E2 -559.81} C_VEL
LIN {X 0,Y 601.39,Z 123.569,A -85,B 0,C 180,E1 -562.684,E2 -562.684} C_VEL
LIN {X 0,Y 601.417,Z 123.568,A -85,B 0,C 180,E1 -565.618,E2 -565.618} C_VEL
LIN {X 0,Y 601.356,Z 123.573,A -85,B 0,C 180,E1 -567.871,E2 -567.871} C_VEL
LIN {X 0,Y 601.388,Z 123.568,A -85,B 0,C 180,E1 -570.166,E2 -570.166} C_VEL
LIN {X 0,Y 601.392,Z 123.572,A -85,B 0,C 180,E1 -572.713,E2 -572.713} C_VEL
LIN {X 0,Y 601.38,Z 123.577,A -85,B 0,C 180,E1 -575.112,E2 -575.112} C_VEL
LIN {X 0,Y 601.425,Z 123.566,A -85,B 0,C 180,E1 -577.42,E2 -577.42} C_VEL
LIN {X 0,Y 601.371,Z 123.57,A -85,B 0,C 180,E1 -579.998,E2 -579.998} C_VEL
LIN {X 0,Y 601.38,Z 123.577,A -85,B 0,C 180,E1 -582.673,E2 -582.673} C_VEL
LIN {X 0,Y 601.393,Z 123.568,A -85,B 0,C 180,E1 -585.48,E2 -585.48} C_VEL
LIN {X 0,Y 601.414,Z 123.571,A -85,B 0,C 180,E1 -588.408,E2 -588.408} C_VEL
LIN {X 0,Y 601.402,Z 123.571,A -85,B 0,C 180,E1 -590.874,E2 -590.874} C_VEL
LIN {X 0,Y 601.389,Z 123.568,A -85,B 0,C 180,E1 -593.417,E2 -593.417} C_VEL
LIN {X 0,Y 601.425,Z 123.568,A -85,B 0,C 180,E1 -596.066,E2 -596.066} C_VEL
LIN {X 0,Y 601.394,Z 123.568,A -85,B 0,C 180,E1 -599.057,E2 -599.057} C_VEL
LIN {X 0,Y 601.396,Z 123.567,A -85,B 0,C 180,E1 -601.372,E2 -601.372} C_VEL
LIN {X 0,Y 601.411,Z 123.575,A -85,B 0,C 180,E1 -604.134,E2 -604.134} C_VEL
LIN {X 0,Y 601.387,Z 123.571,A -85,B 0,C 180,E1 -606.589,E2 -606.589} C_VEL
LIN {X 0,Y 601.407,Z 123.568,A -85,B 0,C 180,E1 -609.478,E2 -609.478} C_VEL
LIN {X 0,Y 601.397,Z 123.66,A -85,B 0,C 180,E1 -611.256,E2 -611.256} C_VEL
LIN {X 0,Y 601.44,Z 135.87,A -85,B 0,C 180,E1 -613.375,E2 -613.375} C_VEL
LIN {X 0,Y 601.432,Z 152.349,A -85,B 0,C 180,E1 -616.197,E2 -616.197} C_VEL
LIN {X 0,Y 601.39,Z 156.326,A -85,B 0,C 180,E1 -616.871,E2 -616.871} C_VEL
LIN {X 0,Y 601.658,Z 162.172,A -85,B 0,C 180,E1 -616.963,E2 -616.963} C_VEL
LIN {X 0,Y 601.623,Z 262.853,A -85,B 0,C 180,E1 -618.183,E2 -618.183} C_VEL
LIN {X 0,Y 601.562,Z 275.392,A -85,B 0,C 180,E1 -618.459,E2 -618.459} C_VEL
LIN {X 0,Y 601.537,Z 288.575,A -85,B 0,C 180,E1 -618.896,E2 -618.896} C_VEL
LIN {X 0,Y 601.514,Z 299.76,A -85,B 0,C 180,E1 -619.396,E2 -619.396} C_VEL
LIN {X 0,Y 601.484,Z 311.531,A -85,B 0,C 180,E1 -620.076,E2 -620.076} C_VEL
LIN {X 0,Y 601.444,Z 322.039,A -85,B 0,C 180,E1 -620.839,E2 -620.839} C_VEL
LIN {X 0,Y 601.429,Z 330.645,A -85,B 0,C 180,E1 -621.601,E2 -621.601} C_VEL
LIN {X 0,Y 601.417,Z 338.572,A -85,B 0,C 180,E1 -622.446,E2 -622.446} C_VEL
LIN {X 0,Y 601.376,Z 345.892,A -85,B 0,C 180,E1 -623.393,E2 -623.393} C_VEL
LIN {X 0,Y 601.372,Z 351.615,A -85,B 0,C 180,E1 -624.3,E2 -624.3} C_VEL
LIN {X 0,Y 601.335,Z 356.755,A -85,B 0,C 180,E1 -625.308,E2 -625.308} C_VEL
LIN {X 0,Y 601.367,Z 360.745,A -85,B 0,C 180,E1 -626.315,E2 -626.315} C_VEL
LIN {X 0,Y 601.324,Z 363.694,A -85,B 0,C 180,E1 -627.321,E2 -627.321} C_VEL
LIN {X 0,Y 601.343,Z 365.127,A -85,B 0,C 180,E1 -627.991,E2 -627.991} C_VEL
LIN {X 0,Y 601.339,Z 366.753,A -85,B 0,C 180,E1 -629.331,E2 -629.331} C_VEL
LIN {X 0,Y 601.336,Z 366.996,A -85,B 0,C 180,E1 -630,E2 -630} C_VEL
LIN {X 0,Y 601.339,Z 366.815,A -85,B 0,C 180,E1 -630.67,E2 -630.67} C_VEL
LIN {X 0,Y 601.344,Z 365.275,A -85,B 0,C 180,E1 -632.01,E2 -632.01} C_VEL
LIN {X 0,Y 601.326,Z 363.916,A -85,B 0,C 180,E1 -632.68,E2 -632.68} C_VEL
LIN {X 0,Y 601.368,Z 361.039,A -85,B 0,C 180,E1 -633.686,E2 -633.686} C_VEL
LIN {X 0,Y 601.337,Z 357.139,A -85,B 0,C 180,E1 -634.693,E2 -634.693} C_VEL
LIN {X 0,Y 601.373,Z 352.108,A -85,B 0,C 180,E1 -635.701,E2 -635.701} C_VEL
LIN {X 0,Y 601.383,Z 345.789,A -85,B 0,C 180,E1 -636.711,E2 -636.711} C_VEL
LIN {X 0,Y 601.396,Z 337.872,A -85,B 0,C 180,E1 -637.724,E2 -637.724} C_VEL
LIN {X 0,Y 601.437,Z 328.027,A -85,B 0,C 180,E1 -638.738,E2 -638.738} C_VEL
LIN {X 0,Y 601.45,Z 317.706,A -85,B 0,C 180,E1 -639.585,E2 -639.585} C_VEL
LIN {X 0,Y 601.481,Z 306.085,A -85,B 0,C 180,E1 -640.35,E2 -640.35} C_VEL
LIN {X 0,Y 601.525,Z 294.194,A -85,B 0,C 180,E1 -640.959,E2 -640.959} C_VEL
LIN {X 0,Y 601.543,Z 281.241,A -85,B 0,C 180,E1 -641.456,E2 -641.456} C_VEL
LIN {X 0,Y 601.609,Z 268.613,A -85,B 0,C 180,E1 -641.797,E2 -641.797} C_VEL
LIN {X 0,Y 601.611,Z 255.481,A -85,B 0,C 180,E1 -642.01,E2 -642.01} C_VEL
LIN {X 0,Y 601.504,Z 157.086,A -85,B 0,C 180,E1 -643.192,E2 -643.192} C_VEL
LIN {X 0,Y 601.402,Z 156.345,A -85,B 0,C 180,E1 -643.215,E2 -643.215} C_VEL
LIN {X 0,Y 601.471,Z 139.369,A -85,B 0,C 180,E1 -646.112,E2 -646.112} C_VEL
LIN {X 0,Y 601.491,Z 124.954,A -85,B 0,C 180,E1 -648.605,E2 -648.605} C_VEL
LIN {X 0,Y 601.401,Z 123.569,A -85,B 0,C 180,E1 -648.868,E2 -648.868} C_VEL
LIN {X 0,Y 601.401,Z 123.567,A -85,B 0,C 180,E1 -651.24,E2 -651.24} C_VEL
LIN {X 0,Y 601.43,Z 123.57,A -85,B 0,C 180,E1 -654.141,E2 -654.141} C_VEL
LIN {X 0,Y 601.387,Z 123.571,A -85,B 0,C 180,E1 -656.364,E2 -656.364} C_VEL
LIN {X 0,Y 601.408,Z 123.565,A -85,B 0,C 180,E1 -658.783,E2 -658.783} C_VEL
LIN {X 0,Y 601.419,Z 123.569,A -85,B 0,C 180,E1 -661.454,E2 -661.454} C_VEL
LIN {X 0,Y 601.419,Z 123.567,A -85,B 0,C 180,E1 -664.119,E2 -664.119} C_VEL
LIN {X 0,Y 601.393,Z 123.567,A -85,B 0,C 180,E1 -666.583,E2 -666.583} C_VEL
LIN {X 0,Y 601.411,Z 123.575,A -85,B 0,C 180,E1 -669.532,E2 -669.532} C_VEL
LIN {X 0,Y 601.408,Z 123.57,A -85,B 0,C 180,E1 -671.766,E2 -671.766} C_VEL
LIN {X 0,Y 601.397,Z 123.567,A -85,B 0,C 180,E1 -674.532,E2 -674.532} C_VEL
LIN {X 0,Y 601.401,Z 123.574,A -85,B 0,C 180,E1 -677.41,E2 -677.41} C_VEL
LIN {X 0,Y 601.377,Z 123.57,A -85,B 0,C 180,E1 -680.002,E2 -680.002} C_VEL
LIN {X 0,Y 601.433,Z 123.564,A -85,B 0,C 180,E1 -682.618,E2 -682.618} C_VEL
LIN {X 0,Y 601.402,Z 123.566,A -85,B 0,C 180,E1 -685.88,E2 -685.88} C_VEL
LIN {X 0,Y 601.412,Z 123.568,A -85,B 0,C 180,E1 -688.546,E2 -688.546} C_VEL
LIN {X 0,Y 601.394,Z 123.57,A -85,B 0,C 180,E1 -691.371,E2 -691.371} C_VEL
LIN {X 0,Y 601.378,Z 123.569,A -85,B 0,C 180,E1 -693.635,E2 -693.635} C_VEL
LIN {X 0,Y 601.395,Z 123.567,A -85,B 0,C 180,E1 -695.857,E2 -695.857} C_VEL
LIN {X 0,Y 601.392,Z 123.576,A -85,B 0,C 180,E1 -698.76,E2 -698.76} C_VEL
LIN {X 0,Y 601.36,Z 123.571,A -85,B 0,C 180,E1 -701.606,E2 -701.606} C_VEL
LIN {X 0,Y 601.391,Z 123.576,A -85,B 0,C 180,E1 -704.408,E2 -704.408} C_VEL
LIN {X 0,Y 601.357,Z 123.572,A -85,B 0,C 180,E1 -707.17,E2 -707.17} C_VEL
LIN {X 0,Y 601.416,Z 123.567,A -85,B 0,C 180,E1 -709.905,E2 -709.905} C_VEL
LIN {X 0,Y 601.373,Z 123.574,A -85,B 0,C 180,E1 -712.614,E2 -712.614} C_VEL
LIN {X 0,Y 601.393,Z 123.571,A -85,B 0,C 180,E1 -714.636,E2 -714.636} C_VEL
LIN {X 0,Y 601.391,Z 123.568,A -85,B 0,C 180,E1 -717.321,E2 -717.321} C_VEL
LIN {X 0,Y 601.439,Z 123.57,A -85,B 0,C 180,E1 -720,E2 -720} C_VEL
LIN {X 0,Y 601.391,Z 123.568,A -85,B 0,C 180,E1 -722.679,E2 -722.679} C_VEL
LIN {X 0,Y 601.383,Z 123.57,A -85,B 0,C 180,E1 -725.364,E2 -725.364} C_VEL
LIN {X 0,Y 601.42,Z 123.57,A -85,B 0,C 180,E1 -728.061,E2 -728.061} C_VEL
LIN {X 0,Y 601.367,Z 123.571,A -85,B 0,C 180,E1 -730.986,E2 -730.986} C_VEL
LIN {X 0,Y 601.379,Z 123.576,A -85,B 0,C 180,E1 -733.517,E2 -733.517} C_VEL
LIN {X 0,Y 601.379,Z 123.57,A -85,B 0,C 180,E1 -736.289,E2 -736.289} C_VEL
LIN {X 0,Y 601.395,Z 123.57,A -85,B 0,C 180,E1 -739.1,E2 -739.1} C_VEL
LIN {X 0,Y 601.372,Z 123.572,A -85,B 0,C 180,E1 -741.961,E2 -741.961} C_VEL
LIN {X 0,Y 601.37,Z 123.573,A -85,B 0,C 180,E1 -744.88,E2 -744.88} C_VEL
LIN {X 0,Y 601.399,Z 123.576,A -85,B 0,C 180,E1 -747.36,E2 -747.36} C_VEL
LIN {X 0,Y 601.367,Z 123.57,A -85,B 0,C 180,E1 -750.168,E2 -750.168} C_VEL
LIN {X 0,Y 601.387,Z 123.571,A -85,B 0,C 180,E1 -752.711,E2 -752.711} C_VEL
LIN {X 0,Y 601.371,Z 123.58,A -85,B 0,C 180,E1 -755.109,E2 -755.109} C_VEL
LIN {X 0,Y 601.428,Z 123.566,A -85,B 0,C 180,E1 -757.42,E2 -757.42} C_VEL
LIN {X 0,Y 601.372,Z 123.57,A -85,B 0,C 180,E1 -759.998,E2 -759.998} C_VEL
LIN {X 0,Y 601.377,Z 123.576,A -85,B 0,C 180,E1 -762.673,E2 -762.673} C_VEL
LIN {X 0,Y 601.398,Z 123.567,A -85,B 0,C 180,E1 -765.48,E2 -765.48} C_VEL
LIN {X 0,Y 601.411,Z 123.57,A -85,B 0,C 180,E1 -768.409,E2 -768.409} C_VEL
LIN {X 0,Y 601.398,Z 123.573,A -85,B 0,C 180,E1 -770.873,E2 -770.873} C_VEL
LIN {X 0,Y 601.388,Z 123.568,A -85,B 0,C 180,E1 -773.416,E2 -773.416} C_VEL
LIN {X 0,Y 601.411,Z 123.568,A -85,B 0,C 180,E1 -776.068,E2 -776.068} C_VEL
LIN {X 0,Y 601.393,Z 123.568,A -85,B 0,C 180,E1 -779.057,E2 -779.057} C_VEL
LIN {X 0,Y 601.394,Z 123.567,A -85,B 0,C 180,E1 -781.371,E2 -781.371} C_VEL
LIN {X 0,Y 601.41,Z 123.574,A -85,B 0,C 180,E1 -784.134,E2 -784.134} C_VEL
LIN {X 0,Y 601.404,Z 123.57,A -85,B 0,C 180,E1 -787.044,E2 -787.044} C_VEL
LIN {X 0,Y 601.379,Z 123.579,A -85,B 0,C 180,E1 -787.134,E2 -787.134} C_VEL
LIN {X 0,Y 601.667,Z 130.051,A -85,B 0,C 180,E1 -788.051,E2 -788.051} C_VEL
LIN {X 0,Y 601.576,Z 149.468,A -85,B 0,C 180,E1 -790.729,E2 -790.729} C_VEL
LIN {X 0,Y 601.522,Z 169.647,A -85,B 0,C 180,E1 -793.469,E2 -793.469} C_VEL
LIN {X 0,Y 601.475,Z 191.077,A -85,B 0,C 180,E1 -796.338,E2 -796.338} C_VEL
LIN {X 0,Y 601.417,Z 194.612,A -85,B 0,C 180,E1 -796.807,E2 -796.807} C_VEL
LIN {X 0,Y 601.658,Z 198.706,A -85,B 0,C 180,E1 -796.876,E2 -796.876} C_VEL
LIN {X 0,Y 601.614,Z 302.937,A -85,B 0,C 180,E1 -798.139,E2 -798.139} C_VEL
LIN {X 0,Y 601.56,Z 316.211,A -85,B 0,C 180,E1 -798.437,E2 -798.437} C_VEL
LIN {X 0,Y 601.546,Z 327.9,A -85,B 0,C 180,E1 -798.825,E2 -798.825} C_VEL
LIN {X 0,Y 601.523,Z 340.629,A -85,B 0,C 180,E1 -799.396,E2 -799.396} C_VEL
LIN {X 0,Y 601.483,Z 352.196,A -85,B 0,C 180,E1 -800.076,E2 -800.076} C_VEL
LIN {X 0,Y 601.444,Z 362.593,A -85,B 0,C 180,E1 -800.839,E2 -800.839} C_VEL
LIN {X 0,Y 601.429,Z 371.11,A -85,B 0,C 180,E1 -801.601,E2 -801.601} C_VEL
LIN {X 0,Y 601.418,Z 378.958,A -85,B 0,C 180,E1 -802.446,E2 -802.446} C_VEL
LIN {X 0,Y 601.37,Z 386.224,A -85,B 0,C 180,E1 -803.398,E2 -803.398} C_VEL
LIN {X 0,Y 601.372,Z 391.865,A -85,B 0,C 180,E1 -804.299,E2 -804.299} C_VEL
LIN {X 0,Y 601.336,Z 396.949,A -85,B 0,C 180,E1 -805.307,E2 -805.307} C_VEL
LIN {X 0,Y 601.368,Z 400.895,A -85,B 0,C 180,E1 -806.314,E2 -806.314} C_VEL
LIN {X 0,Y 601.325,Z 403.808,A -85,B 0,C 180,E1 -807.32,E2 -807.32} C_VEL
LIN {X 0,Y 601.343,Z 405.201,A -85,B 0,C 180,E1 -807.99,E2 -807.99} C_VEL
LIN {X 0,Y 601.339,Z 406.784,A -85,B 0,C 180,E1 -809.33,E2 -809.33} C_VEL
LIN {X 0,Y 601.335,Z 407,A -85,B 0,C 180,E1 -810,E2 -810} C_VEL
LIN {X 0,Y 601.347,Z 406.185,A -85,B 0,C 180,E1 -811.339,E2 -811.339} C_VEL
LIN {X 0,Y 601.343,Z 405.203,A -85,B 0,C 180,E1 -812.009,E2 -812.009} C_VEL
LIN {X 0,Y 601.325,Z 403.81,A -85,B 0,C 180,E1 -812.679,E2 -812.679} C_VEL
LIN {X 0,Y 601.368,Z 400.897,A -85,B 0,C 180,E1 -813.685,E2 -813.685} C_VEL
LIN {X 0,Y 601.336,Z 396.951,A -85,B 0,C 180,E1 -814.692,E2 -814.692} C_VEL
LIN {X 0,Y 601.373,Z 390.88,A -85,B 0,C 180,E1 -815.869,E2 -815.869} C_VEL
LIN {X 0,Y 601.381,Z 384.239,A -85,B 0,C 180,E1 -816.879,E2 -816.879} C_VEL
LIN {X 0,Y 601.4,Z 375.994,A -85,B 0,C 180,E1 -817.892,E2 -817.892} C_VEL
LIN {X 0,Y 601.436,Z 367.542,A -85,B 0,C 180,E1 -818.737,E2 -818.737} C_VEL
LIN {X 0,Y 601.449,Z 357.1,A -85,B 0,C 180,E1 -819.585,E2 -819.585} C_VEL
LIN {X 0,Y 601.467,Z 346.767,A -85,B 0,C 180,E1 -820.264,E2 -820.264} C_VEL
LIN {X 0,Y 601.537,Z 334.601,A -85,B 0,C 180,E1 -820.896,E2 -820.896} C_VEL
LIN {X 0,Y 601.554,Z 322.232,A -85,B 0,C 180,E1 -821.378,E2 -821.378} C_VEL
LIN {X 0,Y 601.582,Z 309.46,A -85,B 0,C 180,E1 -821.732,E2 -821.732} C_VEL
LIN {X 0,Y 601.619,Z 297.125,A -85,B 0,C 180,E1 -821.945,E2 -821.945} C_VEL
LIN {X 0,Y 601.47,Z 195.189,A -85,B 0,C 180,E1 -823.17,E2 -823.17} C_VEL
LIN {X 0,Y 601.455,Z 194.132,A -85,B 0,C 180,E1 -823.256,E2 -823.256} C_VEL
LIN {X 0,Y 601.519,Z 172.773,A -85,B 0,C 180,E1 -826.11,E2 -826.11} C_VEL
LIN {X 0,Y 601.597,Z 150.768,A -85,B 0,C 180,E1 -829.092,E2 -829.092} C_VEL
LIN {X 0,Y 601.651,Z 131.351,A -85,B 0,C 180,E1 -831.769,E2 -831.769} C_VEL
LIN {X 0,Y 601.396,Z 123.584,A -85,B 0,C 180,E1 -832.864,E2 -832.864} C_VEL
LIN {X 0,Y 601.436,Z 123.57,A -85,B 0,C 180,E1 -835.617,E2 -835.617} C_VEL
LIN {X 0,Y 601.384,Z 123.576,A -85,B 0,C 180,E1 -837.868,E2 -837.868} C_VEL
LIN {X 0,Y 601.397,Z 123.569,A -85,B 0,C 180,E1 -840.165,E2 -840.165} C_VEL
LIN {X 0,Y 601.393,Z 123.567,A -85,B 0,C 180,E1 -842.711,E2 -842.711} C_VEL
LIN {X 0,Y 601.378,Z 123.573,A -85,B 0,C 180,E1 -845.109,E2 -845.109} C_VEL
LIN {X 0,Y 601.428,Z 123.573,A -85,B 0,C 180,E1 -847.418,E2 -847.418} C_VEL
LIN {X 0,Y 601.373,Z 123.571,A -85,B 0,C 180,E1 -849.997,E2 -849.997} C_VEL
LIN {X 0,Y 601.373,Z 123.571,A -85,B 0,C 180,E1 -852.672,E2 -852.672} C_VEL
LIN {X 0,Y 601.391,Z 123.573,A -85,B 0,C 180,E1 -855.467,E2 -855.467} C_VEL
LIN {X 0,Y 601.402,Z 123.567,A -85,B 0,C 180,E1 -858.408,E2 -858.408} C_VEL
LIN {X 0,Y 601.392,Z 123.57,A -85,B 0,C 180,E1 -861.532,E2 -861.532} C_VEL
LIN {X 0,Y 601.378,Z 123.57,A -85,B 0,C 180,E1 -863.741,E2 -863.741} C_VEL
LIN {X 0,Y 601.402,Z 123.573,A -85,B 0,C 180,E1 -866.685,E2 -866.685} C_VEL
LIN {X 0,Y 601.387,Z 123.574,A -85,B 0,C 180,E1 -869.056,E2 -869.056} C_VEL
LIN {X 0,Y 601.385,Z 123.57,A -85,B 0,C 180,E1 -871.371,E2 -871.371} C_VEL
LIN {X 0,Y 601.367,Z 123.57,A -85,B 0,C 180,E1 -873.634,E2 -873.634} C_VEL
LIN {X 0,Y 601.388,Z 123.568,A -85,B 0,C 180,E1 -875.857,E2 -875.857} C_VEL
LIN {X 0,Y 601.386,Z 123.575,A -85,B 0,C 180,E1 -878.76,E2 -878.76} C_VEL
LIN {X 0,Y 601.35,Z 123.572,A -85,B 0,C 180,E1 -881.606,E2 -881.606} C_VEL
LIN {X 0,Y 601.381,Z 123.579,A -85,B 0,C 180,E1 -884.408,E2 -884.408} C_VEL
LIN {X 0,Y 601.38,Z 123.577,A -85,B 0,C 180,E1 -886.483,E2 -886.483} C_VEL
LIN {X 0,Y 601.347,Z 123.573,A -85,B 0,C 180,E1 -889.223,E2 -889.223} C_VEL
LIN {X 0,Y 601.417,Z 123.57,A -85,B 0,C 180,E1 -891.939,E2 -891.939} C_VEL
LIN {X 0,Y 601.382,Z 123.571,A -85,B 0,C 180,E1 -894.636,E2 -894.636} C_VEL
LIN {X 0,Y 601.384,Z 123.569,A -85,B 0,C 180,E1 -897.321,E2 -897.321} C_VEL
LIN {X 0,Y 601.434,Z 123.572,A -85,B 0,C 180,E1 -900,E2 -900} C_VEL
LIN {X 0,Y 601.387,Z 123.568,A -85,B 0,C 180,E1 -902.679,E2 -902.679} C_VEL
LIN {X 0,Y 601.39,Z 123.571,A -85,B 0,C 180,E1 -905.364,E2 -905.364} C_VEL
LIN {X 0,Y 601.421,Z 123.569,A -85,B 0,C 180,E1 -908.061,E2 -908.061} C_VEL
LIN {X 0,Y 601.385,Z 123.569,A -85,B 0,C 180,E1 -910.998,E2 -910.998} C_VEL
LIN {X 0,Y 601.369,Z 123.571,A -85,B 0,C 180,E1 -912.334,E2 -912.334} C_VEL
LIN {X 0,Y 600.68,Z 123.657,A -85,B 0,C 180,E1 -912.894,E2 -912.894} C_VEL
LIN {X 0,Y 597.827,Z 124.018,A -85,B 0,C 180,E1 -913.802,E2 -913.802} C_VEL
LIN {X 0,Y 595.431,Z 124.315,A -85,B 0,C 180,E1 -914.532,E2 -914.532} C_VEL
LIN {X 0,Y 594.403,Z 124.441,A -85,B 0,C 180,E1 -915.095,E2 -915.095} C_VEL
LIN {X 0,Y 594.32,Z 124.451,A -85,B 0,C 180,E1 -915.286,E2 -915.286} C_VEL
LIN {X 0,Y 594.317,Z 124.452,A -85,B 0,C 180,E1 -917.906,E2 -917.906} C_VEL
LIN {X 0,Y 594.366,Z 124.444,A -85,B 0,C 180,E1 -920.777,E2 -920.777} C_VEL
LIN {X 0,Y 594.338,Z 124.45,A -85,B 0,C 180,E1 -923.706,E2 -923.706} C_VEL
LIN {X 0,Y 594.34,Z 124.446,A -85,B 0,C 180,E1 -926.016,E2 -926.016} C_VEL
LIN {X 0,Y 594.315,Z 124.449,A -85,B 0,C 180,E1 -928.23,E2 -928.23} C_VEL
LIN {X 0,Y 594.354,Z 124.446,A -85,B 0,C 180,E1 -930.561,E2 -930.561} C_VEL
LIN {X 0,Y 594.364,Z 124.451,A -85,B 0,C 180,E1 -932.951,E2 -932.951} C_VEL
LIN {X 0,Y 594.337,Z 124.45,A -85,B 0,C 180,E1 -935.41,E2 -935.41} C_VEL
LIN {X 0,Y 594.361,Z 124.443,A -85,B 0,C 180,E1 -937.943,E2 -937.943} C_VEL
LIN {X 0,Y 594.366,Z 124.453,A -85,B 0,C 180,E1 -940.822,E2 -940.822} C_VEL
LIN {X 0,Y 594.336,Z 124.446,A -85,B 0,C 180,E1 -943.838,E2 -943.838} C_VEL
LIN {X 0,Y 594.354,Z 124.454,A -85,B 0,C 180,E1 -946.701,E2 -946.701} C_VEL
LIN {X 0,Y 594.356,Z 124.444,A -85,B 0,C 180,E1 -949.433,E2 -949.433} C_VEL
LIN {X 0,Y 594.381,Z 124.449,A -85,B 0,C 180,E1 -952.393,E2 -952.393} C_VEL
LIN {X 0,Y 594.364,Z 124.443,A -85,B 0,C 180,E1 -955.42,E2 -955.42} C_VEL
LIN {X 0,Y 594.369,Z 124.452,A -85,B 0,C 180,E1 -958.359,E2 -958.359} C_VEL
LIN {X 0,Y 594.371,Z 124.442,A -85,B 0,C 180,E1 -961.045,E2 -961.045} C_VEL
LIN {X 0,Y 594.361,Z 124.443,A -85,B 0,C 180,E1 -963.3,E2 -963.3} C_VEL
LIN {X 0,Y 594.349,Z 124.446,A -85,B 0,C 180,E1 -965.575,E2 -965.575} C_VEL
LIN {X 0,Y 594.356,Z 124.448,A -85,B 0,C 180,E1 -968.497,E2 -968.497} C_VEL
LIN {X 0,Y 594.376,Z 124.465,A -85,B 0,C 180,E1 -971.168,E2 -971.168} C_VEL
LIN {X 0,Y 594.424,Z 135.427,A -85,B 0,C 180,E1 -973.095,E2 -973.095} C_VEL
LIN {X 0,Y 594.417,Z 151.117,A -85,B 0,C 180,E1 -975.817,E2 -975.817} C_VEL
LIN {X 0,Y 594.375,Z 156.424,A -85,B 0,C 180,E1 -976.73,E2 -976.73} C_VEL
LIN {X 0,Y 594.744,Z 162.217,A -85,B 0,C 180,E1 -976.809,E2 -976.809} C_VEL
LIN {X 0,Y 594.679,Z 262.882,A -85,B 0,C 180,E1 -978.043,E2 -978.043} C_VEL
LIN {X 0,Y 594.614,Z 275.41,A -85,B 0,C 180,E1 -978.323,E2 -978.323} C_VEL
LIN {X 0,Y 594.563,Z 288.059,A -85,B 0,C 180,E1 -978.743,E2 -978.743} C_VEL
LIN {X 0,Y 594.53,Z 299.774,A -85,B 0,C 180,E1 -979.27,E2 -979.27} C_VEL
LIN {X 0,Y 594.479,Z 311.538,A -85,B 0,C 180,E1 -979.958,E2 -979.958} C_VEL
LIN {X 0,Y 594.414,Z 322.048,A -85,B 0,C 180,E1 -980.73,E2 -980.73} C_VEL
LIN {X 0,Y 594.384,Z 330.651,A -85,B 0,C 180,E1 -981.501,E2 -981.501} C_VEL
LIN {X 0,Y 594.347,Z 338.577,A -85,B 0,C 180,E1 -982.356,E2 -982.356} C_VEL
LIN {X 0,Y 594.305,Z 346.397,A -85,B 0,C 180,E1 -983.39,E2 -983.39} C_VEL
LIN {X 0,Y 594.289,Z 353.443,A -85,B 0,C 180,E1 -984.572,E2 -984.572} C_VEL
LIN {X 0,Y 594.27,Z 358.185,A -85,B 0,C 180,E1 -985.592,E2 -985.592} C_VEL
LIN {X 0,Y 594.267,Z 361.818,A -85,B 0,C 180,E1 -986.61,E2 -986.61} C_VEL
LIN {X 0,Y 594.225,Z 363.696,A -85,B 0,C 180,E1 -987.289,E2 -987.289} C_VEL
LIN {X 0,Y 594.242,Z 365.127,A -85,B 0,C 180,E1 -987.967,E2 -987.967} C_VEL
LIN {X 0,Y 594.24,Z 366.754,A -85,B 0,C 180,E1 -989.323,E2 -989.323} C_VEL
LIN {X 0,Y 594.236,Z 366.996,A -85,B 0,C 180,E1 -990,E2 -990} C_VEL
LIN {X 0,Y 594.239,Z 366.815,A -85,B 0,C 180,E1 -990.678,E2 -990.678} C_VEL
LIN {X 0,Y 594.242,Z 365.275,A -85,B 0,C 180,E1 -992.034,E2 -992.034} C_VEL
LIN {X 0,Y 594.226,Z 363.914,A -85,B 0,C 180,E1 -992.712,E2 -992.712} C_VEL
LIN {X 0,Y 594.289,Z 361.037,A -85,B 0,C 180,E1 -993.73,E2 -993.73} C_VEL
LIN {X 0,Y 594.241,Z 357.137,A -85,B 0,C 180,E1 -994.749,E2 -994.749} C_VEL
LIN {X 0,Y 594.3,Z 352.106,A -85,B 0,C 180,E1 -995.769,E2 -995.769} C_VEL
LIN {X 0,Y 594.316,Z 345.786,A -85,B 0,C 180,E1 -996.792,E2 -996.792} C_VEL
LIN {X 0,Y 594.347,Z 337.868,A -85,B 0,C 180,E1 -997.816,E2 -997.816} C_VEL
LIN {X 0,Y 594.381,Z 328.021,A -85,B 0,C 180,E1 -998.842,E2 -998.842} C_VEL
LIN {X 0,Y 594.432,Z 317.701,A -85,B 0,C 180,E1 -999.7,E2 -999.7} C_VEL
LIN {X 0,Y 594.491,Z 306.073,A -85,B 0,C 180,E1 -1000.473,E2 -1000.473} C_VEL
LIN {X 0,Y 594.55,Z 294.156,A -85,B 0,C 180,E1 -1001.09,E2 -1001.09} C_VEL
LIN {X 0,Y 594.579,Z 281.226,A -85,B 0,C 180,E1 -1001.592,E2 -1001.592} C_VEL
LIN {X 0,Y 594.657,Z 268.589,A -85,B 0,C 180,E1 -1001.937,E2 -1001.937} C_VEL
LIN {X 0,Y 594.693,Z 255.436,A -85,B 0,C 180,E1 -1002.152,E2 -1002.152} C_VEL
LIN {X 0,Y 594.667,Z 158.139,A -85,B 0,C 180,E1 -1003.333,E2 -1003.333} C_VEL
LIN {X 0,Y 594.384,Z 156.342,A -85,B 0,C 180,E1 -1003.374,E2 -1003.374} C_VEL
LIN {X 0,Y 594.459,Z 139.365,A -85,B 0,C 180,E1 -1006.307,E2 -1006.307} C_VEL
LIN {X 0,Y 594.489,Z 126.189,A -85,B 0,C 180,E1 -1008.614,E2 -1008.614} C_VEL
LIN {X 0,Y 594.394,Z 124.443,A -85,B 0,C 180,E1 -1008.945,E2 -1008.945} C_VEL
LIN {X 0,Y 594.36,Z 124.446,A -85,B 0,C 180,E1 -1011.504,E2 -1011.504} C_VEL
LIN {X 0,Y 594.369,Z 124.445,A -85,B 0,C 180,E1 -1014.447,E2 -1014.447} C_VEL
LIN {X 0,Y 594.364,Z 124.443,A -85,B 0,C 180,E1 -1016.7,E2 -1016.7} C_VEL
LIN {X 0,Y 594.374,Z 124.442,A -85,B 0,C 180,E1 -1018.999,E2 -1018.999} C_VEL
LIN {X 0,Y 594.374,Z 124.45,A -85,B 0,C 180,E1 -1021.642,E2 -1021.642} C_VEL
LIN {X 0,Y 594.369,Z 124.442,A -85,B 0,C 180,E1 -1024.581,E2 -1024.581} C_VEL
LIN {X 0,Y 594.385,Z 124.45,A -85,B 0,C 180,E1 -1027.607,E2 -1027.607} C_VEL
LIN {X 0,Y 594.36,Z 124.443,A -85,B 0,C 180,E1 -1030.567,E2 -1030.567} C_VEL
LIN {X 0,Y 594.358,Z 124.452,A -85,B 0,C 180,E1 -1033.3,E2 -1033.3} C_VEL
LIN {X 0,Y 594.341,Z 124.446,A -85,B 0,C 180,E1 -1036.163,E2 -1036.163} C_VEL
LIN {X 0,Y 594.367,Z 124.443,A -85,B 0,C 180,E1 -1038.535,E2 -1038.535} C_VEL
LIN {X 0,Y 594.366,Z 124.451,A -85,B 0,C 180,E1 -1041.297,E2 -1041.297} C_VEL
LIN {X 0,Y 594.34,Z 124.447,A -85,B 0,C 180,E1 -1043.754,E2 -1043.754} C_VEL
LIN {X 0,Y 594.349,Z 124.445,A -85,B 0,C 180,E1 -1046.237,E2 -1046.237} C_VEL
LIN {X 0,Y 594.36,Z 124.448,A -85,B 0,C 180,E1 -1048.649,E2 -1048.649} C_VEL
LIN {X 0,Y 594.368,Z 124.45,A -85,B 0,C 180,E1 -1051.044,E2 -1051.044} C_VEL
LIN {X 0,Y 594.371,Z 124.445,A -85,B 0,C 180,E1 -1053.3,E2 -1053.3} C_VEL
LIN {X 0,Y 594.332,Z 124.447,A -85,B 0,C 180,E1 -1055.577,E2 -1055.577} C_VEL
LIN {X 0,Y 594.35,Z 124.451,A -85,B 0,C 180,E1 -1058.496,E2 -1058.496} C_VEL
LIN {X 0,Y 594.341,Z 124.446,A -85,B 0,C 180,E1 -1061.381,E2 -1061.381} C_VEL
LIN {X 0,Y 594.337,Z 124.451,A -85,B 0,C 180,E1 -1064.218,E2 -1064.218} C_VEL
LIN {X 0,Y 594.312,Z 124.451,A -85,B 0,C 180,E1 -1067.016,E2 -1067.016} C_VEL
LIN {X 0,Y 594.371,Z 124.444,A -85,B 0,C 180,E1 -1069.784,E2 -1069.784} C_VEL
LIN {X 0,Y 594.346,Z 124.451,A -85,B 0,C 180,E1 -1072.526,E2 -1072.526} C_VEL
LIN {X 0,Y 594.344,Z 124.445,A -85,B 0,C 180,E1 -1075.252,E2 -1075.252} C_VEL
LIN {X 0,Y 594.399,Z 124.446,A -85,B 0,C 180,E1 -1077.967,E2 -1077.967} C_VEL
LIN {X 0,Y 594.318,Z 124.45,A -85,B 0,C 180,E1 -1080.678,E2 -1080.678} C_VEL
LIN {X 0,Y 594.359,Z 124.444,A -85,B 0,C 180,E1 -1082.711,E2 -1082.711} C_VEL
LIN {X 0,Y 594.353,Z 124.447,A -85,B 0,C 180,E1 -1085.428,E2 -1085.428} C_VEL
LIN {X 0,Y 594.363,Z 124.448,A -85,B 0,C 180,E1 -1088.157,E2 -1088.157} C_VEL
LIN {X 0,Y 594.325,Z 124.448,A -85,B 0,C 180,E1 -1091.044,E2 -1091.044} C_VEL
LIN {X 0,Y 594.348,Z 124.455,A -85,B 0,C 180,E1 -1093.68,E2 -1093.68} C_VEL
LIN {X 0,Y 594.31,Z 124.449,A -85,B 0,C 180,E1 -1096.693,E2 -1096.693} C_VEL
LIN {X 0,Y 594.346,Z 124.452,A -85,B 0,C 180,E1 -1099.335,E2 -1099.335} C_VEL
LIN {X 0,Y 594.341,Z 124.455,A -85,B 0,C 180,E1 -1101.504,E2 -1101.504} C_VEL
LIN {X 0,Y 594.336,Z 124.446,A -85,B 0,C 180,E1 -1104.448,E2 -1104.448} C_VEL
LIN {X 0,Y 594.352,Z 124.446,A -85,B 0,C 180,E1 -1106.701,E2 -1106.701} C_VEL
LIN {X 0,Y 594.33,Z 124.449,A -85,B 0,C 180,E1 -1109.779,E2 -1109.779} C_VEL
LIN {X 0,Y 594.334,Z 124.446,A -85,B 0,C 180,E1 -1112.149,E2 -1112.149} C_VEL
LIN {X 0,Y 594.355,Z 124.446,A -85,B 0,C 180,E1 -1114.582,E2 -1114.582} C_VEL
LIN {X 0,Y 594.378,Z 124.443,A -85,B 0,C 180,E1 -1117.607,E2 -1117.607} C_VEL
LIN {X 0,Y 594.356,Z 124.448,A -85,B 0,C 180,E1 -1120.568,E2 -1120.568} C_VEL
LIN {X 0,Y 594.341,Z 124.449,A -85,B 0,C 180,E1 -1123.302,E2 -1123.302} C_VEL
LIN {X 0,Y 594.342,Z 124.447,A -85,B 0,C 180,E1 -1126.163,E2 -1126.163} C_VEL
LIN {X 0,Y 594.361,Z 124.446,A -85,B 0,C 180,E1 -1129.18,E2 -1129.18} C_VEL
LIN {X 0,Y 594.351,Z 124.447,A -85,B 0,C 180,E1 -1132.057,E2 -1132.057} C_VEL
LIN {X 0,Y 594.324,Z 124.455,A -85,B 0,C 180,E1 -1134.681,E2 -1134.681} C_VEL
LIN {X 0,Y 594.37,Z 124.443,A -85,B 0,C 180,E1 -1137.09,E2 -1137.09} C_VEL
LIN {X 0,Y 594.365,Z 124.444,A -85,B 0,C 180,E1 -1139.676,E2 -1139.676} C_VEL
LIN {X 0,Y 594.377,Z 124.448,A -85,B 0,C 180,E1 -1142.539,E2 -1142.539} C_VEL
LIN {X 0,Y 594.368,Z 124.445,A -85,B 0,C 180,E1 -1144.807,E2 -1144.807} C_VEL
LIN {X 0,Y 594.389,Z 124.55,A -85,B 0,C 180,E1 -1146.988,E2 -1146.988} C_VEL
LIN {X 0,Y 594.757,Z 129.043,A -85,B 0,C 180,E1 -1147.64,E2 -1147.64} C_VEL
LIN {X 0,Y 594.662,Z 149.468,A -85,B 0,C 180,E1 -1150.496,E2 -1150.496} C_VEL
LIN {X 0,Y 594.548,Z 171.473,A -85,B 0,C 180,E1 -1153.519,E2 -1153.519} C_VEL
LIN {X 0,Y 594.425,Z 193.479,A -85,B 0,C 180,E1 -1156.496,E2 -1156.496} C_VEL
LIN {X 0,Y 594.436,Z 194.612,A -85,B 0,C 180,E1 -1156.649,E2 -1156.649} C_VEL
LIN {X 0,Y 594.739,Z 198.706,A -85,B 0,C 180,E1 -1156.721,E2 -1156.721} C_VEL
LIN {X 0,Y 594.666,Z 302.937,A -85,B 0,C 180,E1 -1157.999,E2 -1157.999} C_VEL
LIN {X 0,Y 594.601,Z 316.212,A -85,B 0,C 180,E1 -1158.3,E2 -1158.3} C_VEL
LIN {X 0,Y 594.577,Z 328.484,A -85,B 0,C 180,E1 -1158.715,E2 -1158.715} C_VEL
LIN {X 0,Y 594.536,Z 340.628,A -85,B 0,C 180,E1 -1159.27,E2 -1159.27} C_VEL
LIN {X 0,Y 594.477,Z 352.198,A -85,B 0,C 180,E1 -1159.957,E2 -1159.957} C_VEL
LIN {X 0,Y 594.414,Z 362.595,A -85,B 0,C 180,E1 -1160.729,E2 -1160.729} C_VEL
LIN {X 0,Y 594.383,Z 371.11,A -85,B 0,C 180,E1 -1161.5,E2 -1161.5} C_VEL
LIN {X 0,Y 594.347,Z 378.958,A -85,B 0,C 180,E1 -1162.355,E2 -1162.355} C_VEL
LIN {X 0,Y 594.283,Z 386.812,A -85,B 0,C 180,E1 -1163.408,E2 -1163.408} C_VEL
LIN {X 0,Y 594.289,Z 393.679,A -85,B 0,C 180,E1 -1164.571,E2 -1164.571} C_VEL
LIN {X 0,Y 594.27,Z 398.37,A -85,B 0,C 180,E1 -1165.591,E2 -1165.591} C_VEL
LIN {X 0,Y 594.267,Z 401.956,A -85,B 0,C 180,E1 -1166.61,E2 -1166.61} C_VEL
LIN {X 0,Y 594.225,Z 403.808,A -85,B 0,C 180,E1 -1167.288,E2 -1167.288} C_VEL
LIN {X 0,Y 594.242,Z 405.2,A -85,B 0,C 180,E1 -1167.966,E2 -1167.966} C_VEL
LIN {X 0,Y 594.239,Z 406.784,A -85,B 0,C 180,E1 -1169.322,E2 -1169.322} C_VEL
LIN {X 0,Y 594.236,Z 407,A -85,B 0,C 180,E1 -1170,E2 -1170} C_VEL
LIN {X 0,Y 594.247,Z 406.185,A -85,B 0,C 180,E1 -1171.355,E2 -1171.355} C_VEL
LIN {X 0,Y 594.242,Z 405.202,A -85,B 0,C 180,E1 -1172.033,E2 -1172.033} C_VEL
LIN {X 0,Y 594.226,Z 403.811,A -85,B 0,C 180,E1 -1172.711,E2 -1172.711} C_VEL
LIN {X 0,Y 594.289,Z 400.897,A -85,B 0,C 180,E1 -1173.729,E2 -1173.729} C_VEL
LIN {X 0,Y 594.241,Z 396.951,A -85,B 0,C 180,E1 -1174.748,E2 -1174.748} C_VEL
LIN {X 0,Y 594.305,Z 390.88,A -85,B 0,C 180,E1 -1175.939,E2 -1175.939} C_VEL
LIN {X 0,Y 594.307,Z 384.24,A -85,B 0,C 180,E1 -1176.962,E2 -1176.962} C_VEL
LIN {X 0,Y 594.359,Z 375.994,A -85,B 0,C 180,E1 -1177.986,E2 -1177.986} C_VEL
LIN {X 0,Y 594.382,Z 367.543,A -85,B 0,C 180,E1 -1178.842,E2 -1178.842} C_VEL
LIN {X 0,Y 594.432,Z 357.102,A -85,B 0,C 180,E1 -1179.699,E2 -1179.699} C_VEL
LIN {X 0,Y 594.481,Z 346.767,A -85,B 0,C 180,E1 -1180.386,E2 -1180.386} C_VEL
LIN {X 0,Y 594.557,Z 335.725,A -85,B 0,C 180,E1 -1180.973,E2 -1180.973} C_VEL
LIN {X 0,Y 594.578,Z 323.724,A -85,B 0,C 180,E1 -1181.464,E2 -1181.464} C_VEL
LIN {X 0,Y 594.624,Z 310.373,A -85,B 0,C 180,E1 -1181.85,E2 -1181.85} C_VEL
LIN {X 0,Y 594.699,Z 297.125,A -85,B 0,C 180,E1 -1182.086,E2 -1182.086} C_VEL
LIN {X 0,Y 594.617,Z 196.307,A -85,B 0,C 180,E1 -1183.311,E2 -1183.311} C_VEL
LIN {X 0,Y 594.436,Z 194.617,A -85,B 0,C 180,E1 -1183.351,E2 -1183.351} C_VEL
LIN {X 0,Y 594.518,Z 172.773,A -85,B 0,C 180,E1 -1186.305,E2 -1186.305} C_VEL
LIN {X 0,Y 594.628,Z 152.412,A -85,B 0,C 180,E1 -1189.097,E2 -1189.097} C_VEL
LIN {X 0,Y 594.751,Z 131.351,A -85,B 0,C 180,E1 -1192.035,E2 -1192.035} C_VEL
LIN {X 0,Y 594.624,Z 126.018,A -85,B 0,C 180,E1 -1192.794,E2 -1192.794} C_VEL
LIN {X 0,Y 594.375,Z 124.447,A -85,B 0,C 180,E1 -1193.058,E2 -1193.058} C_VEL
LIN {X 0,Y 594.36,Z 124.45,A -85,B 0,C 180,E1 -1196.017,E2 -1196.017} C_VEL
LIN {X 0,Y 594.35,Z 124.447,A -85,B 0,C 180,E1 -1198.227,E2 -1198.227} C_VEL
LIN {X 0,Y 594.36,Z 124.444,A -85,B 0,C 180,E1 -1200.56,E2 -1200.56} C_VEL
LIN {X 0,Y 594.37,Z 124.444,A -85,B 0,C 180,E1 -1202.95,E2 -1202.95} C_VEL
LIN {X 0,Y 594.322,Z 124.457,A -85,B 0,C 180,E1 -1205.41,E2 -1205.41} C_VEL
LIN {X 0,Y 594.362,Z 124.445,A -85,B 0,C 180,E1 -1207.941,E2 -1207.941} C_VEL
LIN {X 0,Y 594.369,Z 124.444,A -85,B 0,C 180,E1 -1210.821,E2 -1210.821} C_VEL
LIN {X 0,Y 594.353,Z 124.446,A -85,B 0,C 180,E1 -1213.838,E2 -1213.838} C_VEL
LIN {X 0,Y 594.338,Z 124.449,A -85,B 0,C 180,E1 -1216.698,E2 -1216.698} C_VEL
LIN {X 0,Y 594.352,Z 124.449,A -85,B 0,C 180,E1 -1219.431,E2 -1219.431} C_VEL
LIN {X 0,Y 594.375,Z 124.443,A -85,B 0,C 180,E1 -1222.392,E2 -1222.392} C_VEL
LIN {X 0,Y 594.356,Z 124.446,A -85,B 0,C 180,E1 -1225.418,E2 -1225.418} C_VEL
LIN {X 0,Y 594.358,Z 124.446,A -85,B 0,C 180,E1 -1228.358,E2 -1228.358} C_VEL
LIN {X 0,Y 594.361,Z 124.449,A -85,B 0,C 180,E1 -1231.044,E2 -1231.044} C_VEL
LIN {X 0,Y 594.352,Z 124.446,A -85,B 0,C 180,E1 -1233.299,E2 -1233.299} C_VEL
LIN {X 0,Y 594.324,Z 124.448,A -85,B 0,C 180,E1 -1235.577,E2 -1235.577} C_VEL
LIN {X 0,Y 594.342,Z 124.455,A -85,B 0,C 180,E1 -1238.496,E2 -1238.496} C_VEL
LIN {X 0,Y 594.33,Z 124.447,A -85,B 0,C 180,E1 -1241.381,E2 -1241.381} C_VEL
LIN {X 0,Y 594.328,Z 124.454,A -85,B 0,C 180,E1 -1244.218,E2 -1244.218} C_VEL
LIN {X 0,Y 594.346,Z 124.455,A -85,B 0,C 180,E1 -1246.32,E2 -1246.32} C_VEL
LIN {X 0,Y 594.331,Z 124.447,A -85,B 0,C 180,E1 -1249.094,E2 -1249.094} C_VEL
LIN {X 0,Y 594.359,Z 124.448,A -85,B 0,C 180,E1 -1251.843,E2 -1251.843} C_VEL
LIN {X 0,Y 594.352,Z 124.447,A -85,B 0,C 180,E1 -1254.572,E2 -1254.572} C_VEL
LIN {X 0,Y 594.352,Z 124.445,A -85,B 0,C 180,E1 -1257.289,E2 -1257.289} C_VEL
LIN {X 0,Y 594.402,Z 124.448,A -85,B 0,C 180,E1 -1260,E2 -1260} C_VEL
LIN {X 0,Y 594.355,Z 124.444,A -85,B 0,C 180,E1 -1262.711,E2 -1262.711} C_VEL
LIN {X 0,Y 594.36,Z 124.447,A -85,B 0,C 180,E1 -1265.428,E2 -1265.428} C_VEL
LIN {X 0,Y 594.363,Z 124.446,A -85,B 0,C 180,E1 -1268.157,E2 -1268.157} C_VEL
LIN {X 0,Y 594.352,Z 124.446,A -85,B 0,C 180,E1 -1271.061,E2 -1271.061} C_VEL
LIN {X 0,Y 594.352,Z 124.453,A -85,B 0,C 180,E1 -1273.68,E2 -1273.68} C_VEL
LIN {X 0,Y 594.32,Z 124.451,A -85,B 0,C 180,E1 -1275.286,E2 -1275.286} C_VEL
LIN {X 0,Y 593.649,Z 124.538,A -85,B 0,C 180,E1 -1275.852,E2 -1275.852} C_VEL
LIN {X 0,Y 590.784,Z 124.893,A -85,B 0,C 180,E1 -1276.769,E2 -1276.769} C_VEL
LIN {X 0,Y 588.372,Z 125.199,A -85,B 0,C 180,E1 -1277.507,E2 -1277.507} C_VEL
LIN {X 0,Y 587.347,Z 125.319,A -85,B 0,C 180,E1 -1278.077,E2 -1278.077} C_VEL
LIN {X 0,Y 587.27,Z 125.327,A -85,B 0,C 180,E1 -1278.27,E2 -1278.27} C_VEL
LIN {X 0,Y 587.321,Z 125.325,A -85,B 0,C 180,E1 -1281.038,E2 -1281.038} C_VEL
LIN {X 0,Y 587.278,Z 125.326,A -85,B 0,C 180,E1 -1284.009,E2 -1284.009} C_VEL
LIN {X 0,Y 587.295,Z 125.323,A -85,B 0,C 180,E1 -1286.281,E2 -1286.281} C_VEL
LIN {X 0,Y 587.331,Z 125.329,A -85,B 0,C 180,E1 -1289.132,E2 -1289.132} C_VEL
LIN {X 0,Y 587.305,Z 125.323,A -85,B 0,C 180,E1 -1291.831,E2 -1291.831} C_VEL
LIN {X 0,Y 587.327,Z 125.32,A -85,B 0,C 180,E1 -1294.347,E2 -1294.347} C_VEL
LIN {X 0,Y 587.331,Z 125.32,A -85,B 0,C 180,E1 -1297.609,E2 -1297.609} C_VEL
LIN {X 0,Y 587.296,Z 125.325,A -85,B 0,C 180,E1 -1300.256,E2 -1300.256} C_VEL
LIN {X 0,Y 587.288,Z 125.329,A -85,B 0,C 180,E1 -1303.117,E2 -1303.117} C_VEL
LIN {X 0,Y 587.306,Z 125.323,A -85,B 0,C 180,E1 -1306.049,E2 -1306.049} C_VEL
LIN {X 0,Y 587.331,Z 125.324,A -85,B 0,C 180,E1 -1308.926,E2 -1308.926} C_VEL
LIN {X 0,Y 587.31,Z 125.321,A -85,B 0,C 180,E1 -1311.52,E2 -1311.52} C_VEL
LIN {X 0,Y 587.282,Z 125.329,A -85,B 0,C 180,E1 -1314.1,E2 -1314.1} C_VEL
LIN {X 0,Y 587.333,Z 125.321,A -85,B 0,C 180,E1 -1316.89,E2 -1316.89} C_VEL
LIN {X 0,Y 587.317,Z 125.321,A -85,B 0,C 180,E1 -1319.494,E2 -1319.494} C_VEL
LIN {X 0,Y 587.3,Z 125.332,A -85,B 0,C 180,E1 -1322.181,E2 -1322.181} C_VEL
LIN {X 0,Y 587.329,Z 125.324,A -85,B 0,C 180,E1 -1324.484,E2 -1324.484} C_VEL
LIN {X 0,Y 587.308,Z 125.323,A -85,B 0,C 180,E1 -1327.486,E2 -1327.486} C_VEL
LIN {X 0,Y 587.314,Z 125.327,A -85,B 0,C 180,E1 -1329.695,E2 -1329.695} C_VEL
LIN {X 0,Y 587.348,Z 125.418,A -85,B 0,C 180,E1 -1331.104,E2 -1331.104} C_VEL
LIN {X 0,Y 587.406,Z 135.7,A -85,B 0,C 180,E1 -1332.935,E2 -1332.935} C_VEL
LIN {X 0,Y 587.378,Z 151.651,A -85,B 0,C 180,E1 -1335.737,E2 -1335.737} C_VEL
LIN {X 0,Y 587.357,Z 156.455,A -85,B 0,C 180,E1 -1336.568,E2 -1336.568} C_VEL
LIN {X 0,Y 587.866,Z 160.474,A -85,B 0,C 180,E1 -1336.63,E2 -1336.63} C_VEL
LIN {X 0,Y 587.735,Z 262.911,A -85,B 0,C 180,E1 -1337.9,E2 -1337.9} C_VEL
LIN {X 0,Y 587.668,Z 276.189,A -85,B 0,C 180,E1 -1338.205,E2 -1338.205} C_VEL
LIN {X 0,Y 587.611,Z 288.741,A -85,B 0,C 180,E1 -1338.634,E2 -1338.634} C_VEL
LIN {X 0,Y 587.548,Z 299.788,A -85,B 0,C 180,E1 -1339.141,E2 -1339.141} C_VEL
LIN {X 0,Y 587.468,Z 311.543,A -85,B 0,C 180,E1 -1339.837,E2 -1339.837} C_VEL
LIN {X 0,Y 587.394,Z 322.056,A -85,B 0,C 180,E1 -1340.618,E2 -1340.618} C_VEL
LIN {X 0,Y 587.323,Z 330.657,A -85,B 0,C 180,E1 -1341.398,E2 -1341.398} C_VEL
LIN {X 0,Y 587.274,Z 338.581,A -85,B 0,C 180,E1 -1342.263,E2 -1342.263} C_VEL
LIN {X 0,Y 587.235,Z 345.152,A -85,B 0,C 180,E1 -1343.127,E2 -1343.127} C_VEL
LIN {X 0,Y 587.237,Z 351.621,A -85,B 0,C 180,E1 -1344.162,E2 -1344.162} C_VEL
LIN {X 0,Y 587.146,Z 356.76,A -85,B 0,C 180,E1 -1345.194,E2 -1345.194} C_VEL
LIN {X 0,Y 587.213,Z 360.749,A -85,B 0,C 180,E1 -1346.226,E2 -1346.226} C_VEL
LIN {X 0,Y 587.131,Z 363.698,A -85,B 0,C 180,E1 -1347.256,E2 -1347.256} C_VEL
LIN {X 0,Y 587.141,Z 365.127,A -85,B 0,C 180,E1 -1347.942,E2 -1347.942} C_VEL
LIN {X 0,Y 587.14,Z 366.754,A -85,B 0,C 180,E1 -1349.315,E2 -1349.315} C_VEL
LIN {X 0,Y 587.137,Z 366.996,A -85,B 0,C 180,E1 -1350,E2 -1350} C_VEL
LIN {X 0,Y 587.14,Z 366.815,A -85,B 0,C 180,E1 -1350.686,E2 -1350.686} C_VEL
LIN {X 0,Y 587.141,Z 365.272,A -85,B 0,C 180,E1 -1352.058,E2 -1352.058} C_VEL
LIN {X 0,Y 587.133,Z 363.911,A -85,B 0,C 180,E1 -1352.745,E2 -1352.745} C_VEL
LIN {X 0,Y 587.213,Z 361.035,A -85,B 0,C 180,E1 -1353.775,E2 -1353.775} C_VEL
LIN {X 0,Y 587.147,Z 357.135,A -85,B 0,C 180,E1 -1354.807,E2 -1354.807} C_VEL
LIN {X 0,Y 587.23,Z 352.103,A -85,B 0,C 180,E1 -1355.839,E2 -1355.839} C_VEL
LIN {X 0,Y 587.231,Z 345.782,A -85,B 0,C 180,E1 -1356.874,E2 -1356.874} C_VEL
LIN {X 0,Y 587.288,Z 337.863,A -85,B 0,C 180,E1 -1357.91,E2 -1357.91} C_VEL
LIN {X 0,Y 587.343,Z 328.014,A -85,B 0,C 180,E1 -1358.949,E2 -1358.949} C_VEL
LIN {X 0,Y 587.419,Z 317.696,A -85,B 0,C 180,E1 -1359.817,E2 -1359.817} C_VEL
LIN {X 0,Y 587.497,Z 306.062,A -85,B 0,C 180,E1 -1360.599,E2 -1360.599} C_VEL
LIN {X 0,Y 587.569,Z 295.113,A -85,B 0,C 180,E1 -1361.18,E2 -1361.18} C_VEL
LIN {X 0,Y 587.625,Z 282.451,A -85,B 0,C 180,E1 -1361.69,E2 -1361.69} C_VEL
LIN {X 0,Y 587.715,Z 269.481,A -85,B 0,C 180,E1 -1362.058,E2 -1362.058} C_VEL
LIN {X 0,Y 587.776,Z 257.158,A -85,B 0,C 180,E1 -1362.275,E2 -1362.275} C_VEL
LIN {X 0,Y 587.691,Z 158.785,A -85,B 0,C 180,E1 -1363.485,E2 -1363.485} C_VEL
LIN {X 0,Y 587.366,Z 156.339,A -85,B 0,C 180,E1 -1363.537,E2 -1363.537} C_VEL
LIN {X 0,Y 587.432,Z 139.362,A -85,B 0,C 180,E1 -1366.508,E2 -1366.508} C_VEL
LIN {X 0,Y 587.42,Z 126.185,A -85,B 0,C 180,E1 -1368.847,E2 -1368.847} C_VEL
LIN {X 0,Y 587.348,Z 125.321,A -85,B 0,C 180,E1 -1369.04,E2 -1369.04} C_VEL
LIN {X 0,Y 587.315,Z 125.328,A -85,B 0,C 180,E1 -1371.775,E2 -1371.775} C_VEL
LIN {X 0,Y 587.315,Z 125.321,A -85,B 0,C 180,E1 -1374.76,E2 -1374.76} C_VEL
LIN {X 0,Y 587.306,Z 125.329,A -85,B 0,C 180,E1 -1377.684,E2 -1377.684} C_VEL
LIN {X 0,Y 587.316,Z 125.325,A -85,B 0,C 180,E1 -1380.171,E2 -1380.171} C_VEL
LIN {X 0,Y 587.329,Z 125.319,A -85,B 0,C 180,E1 -1382.579,E2 -1382.579} C_VEL
LIN {X 0,Y 587.32,Z 125.322,A -85,B 0,C 180,E1 -1385.056,E2 -1385.056} C_VEL
LIN {X 0,Y 587.33,Z 125.325,A -85,B 0,C 180,E1 -1387.837,E2 -1387.837} C_VEL
LIN {X 0,Y 587.305,Z 125.323,A -85,B 0,C 180,E1 -1390.255,E2 -1390.255} C_VEL
LIN {X 0,Y 587.3,Z 125.328,A -85,B 0,C 180,E1 -1393.116,E2 -1393.116} C_VEL
LIN {X 0,Y 587.297,Z 125.324,A -85,B 0,C 180,E1 -1396.047,E2 -1396.047} C_VEL
LIN {X 0,Y 587.33,Z 125.324,A -85,B 0,C 180,E1 -1398.925,E2 -1398.925} C_VEL
LIN {X 0,Y 587.313,Z 125.326,A -85,B 0,C 180,E1 -1401.519,E2 -1401.519} C_VEL
LIN {X 0,Y 587.276,Z 125.326,A -85,B 0,C 180,E1 -1404.099,E2 -1404.099} C_VEL
LIN {X 0,Y 587.33,Z 125.327,A -85,B 0,C 180,E1 -1406.889,E2 -1406.889} C_VEL
LIN {X 0,Y 587.304,Z 125.324,A -85,B 0,C 180,E1 -1409.495,E2 -1409.495} C_VEL
LIN {X 0,Y 587.287,Z 125.327,A -85,B 0,C 180,E1 -1411.401,E2 -1411.401} C_VEL
LIN {X 0,Y 587.328,Z 125.319,A -85,B 0,C 180,E1 -1413.824,E2 -1413.824} C_VEL
LIN {X 0,Y 587.296,Z 125.334,A -85,B 0,C 180,E1 -1416.74,E2 -1416.74} C_VEL
LIN {X 0,Y 587.328,Z 125.325,A -85,B 0,C 180,E1 -1418.962,E2 -1418.962} C_VEL
LIN {X 0,Y 587.273,Z 125.327,A -85,B 0,C 180,E1 -1421.872,E2 -1421.872} C_VEL
LIN {X 0,Y 587.297,Z 125.329,A -85,B 0,C 180,E1 -1424.736,E2 -1424.736} C_VEL
LIN {X 0,Y 587.269,Z 125.33,A -85,B 0,C 180,E1 -1426.857,E2 -1426.857} C_VEL
LIN {X 0,Y 587.322,Z 125.321,A -85,B 0,C 180,E1 -1429.66,E2 -1429.66} C_VEL
LIN {X 0,Y 587.307,Z 125.329,A -85,B 0,C 180,E1 -1432.436,E2 -1432.436} C_VEL
LIN {X 0,Y 587.318,Z 125.32,A -85,B 0,C 180,E1 -1435.195,E2 -1435.195} C_VEL
LIN {X 0,Y 587.367,Z 125.321,A -85,B 0,C 180,E1 -1437.943,E2 -1437.943} C_VEL
LIN {X 0,Y 587.375,Z 125.322,A -85,B 0,C 180,E1 -1440,E2 -1440} C_VEL
LIN {X 0,Y 587.328,Z 125.32,A -85,B 0,C 180,E1 -1442.743,E2 -1442.743} C_VEL
LIN {X 0,Y 587.323,Z 125.323,A -85,B 0,C 180,E1 -1445.493,E2 -1445.493} C_VEL
LIN {X 0,Y 587.319,Z 125.324,A -85,B 0,C 180,E1 -1448.256,E2 -1448.256} C_VEL
LIN {X 0,Y 587.292,Z 125.325,A -85,B 0,C 180,E1 -1451.107,E2 -1451.107} C_VEL
LIN {X 0,Y 587.311,Z 125.323,A -85,B 0,C 180,E1 -1454.241,E2 -1454.241} C_VEL
LIN {X 0,Y 587.287,Z 125.325,A -85,B 0,C 180,E1 -1456.796,E2 -1456.796} C_VEL
LIN {X 0,Y 587.289,Z 125.333,A -85,B 0,C 180,E1 -1459.577,E2 -1459.577} C_VEL
LIN {X 0,Y 587.289,Z 125.329,A -85,B 0,C 180,E1 -1461.776,E2 -1461.776} C_VEL
LIN {X 0,Y 587.292,Z 125.325,A -85,B 0,C 180,E1 -1464.761,E2 -1464.761} C_VEL
LIN {X 0,Y 587.291,Z 125.328,A -85,B 0,C 180,E1 -1467.682,E2 -1467.682} C_VEL
LIN {X 0,Y 587.284,Z 125.326,A -85,B 0,C 180,E1 -1470.502,E2 -1470.502} C_VEL
LIN {X 0,Y 587.315,Z 125.326,A -85,B 0,C 180,E1 -1473.398,E2 -1473.398} C_VEL
LIN {X 0,Y 587.27,Z 125.327,A -85,B 0,C 180,E1 -1475.902,E2 -1475.902} C_VEL
LIN {X 0,Y 587.309,Z 125.324,A -85,B 0,C 180,E1 -1478.481,E2 -1478.481} C_VEL
LIN {X 0,Y 587.328,Z 125.325,A -85,B 0,C 180,E1 -1481.158,E2 -1481.158} C_VEL
LIN {X 0,Y 587.3,Z 125.323,A -85,B 0,C 180,E1 -1484.111,E2 -1484.111} C_VEL
LIN {X 0,Y 587.286,Z 125.33,A -85,B 0,C 180,E1 -1486.991,E2 -1486.991} C_VEL
LIN {X 0,Y 587.292,Z 125.324,A -85,B 0,C 180,E1 -1489.744,E2 -1489.744} C_VEL
LIN {X 0,Y 587.332,Z 125.325,A -85,B 0,C 180,E1 -1492.392,E2 -1492.392} C_VEL
LIN {X 0,Y 587.328,Z 125.319,A -85,B 0,C 180,E1 -1495.656,E2 -1495.656} C_VEL
LIN {X 0,Y 587.332,Z 125.326,A -85,B 0,C 180,E1 -1498.231,E2 -1498.231} C_VEL
LIN {X 0,Y 587.341,Z 125.32,A -85,B 0,C 180,E1 -1500.869,E2 -1500.869} C_VEL
LIN {X 0,Y 587.31,Z 125.326,A -85,B 0,C 180,E1 -1503.829,E2 -1503.829} C_VEL
LIN {X 0,Y 587.317,Z 125.409,A -85,B 0,C 180,E1 -1506.847,E2 -1506.847} C_VEL
LIN {X 0,Y 587.834,Z 129.954,A -85,B 0,C 180,E1 -1507.506,E2 -1507.506} C_VEL
LIN {X 0,Y 587.74,Z 149.468,A -85,B 0,C 180,E1 -1510.257,E2 -1510.257} C_VEL
LIN {X 0,Y 587.525,Z 170.129,A -85,B 0,C 180,E1 -1513.13,E2 -1513.13} C_VEL
LIN {X 0,Y 587.451,Z 189.887,A -85,B 0,C 180,E1 -1515.843,E2 -1515.843} C_VEL
LIN {X 0,Y 587.381,Z 194.612,A -85,B 0,C 180,E1 -1516.485,E2 -1516.485} C_VEL
LIN {X 0,Y 587.838,Z 198.706,A -85,B 0,C 180,E1 -1516.562,E2 -1516.562} C_VEL
LIN {X 0,Y 587.724,Z 302.937,A -85,B 0,C 180,E1 -1517.855,E2 -1517.855} C_VEL
LIN {X 0,Y 587.668,Z 316.213,A -85,B 0,C 180,E1 -1518.16,E2 -1518.16} C_VEL
LIN {X 0,Y 587.606,Z 328.637,A -85,B 0,C 180,E1 -1518.585,E2 -1518.585} C_VEL
LIN {X 0,Y 587.557,Z 340.626,A -85,B 0,C 180,E1 -1519.141,E2 -1519.141} C_VEL
LIN {X 0,Y 587.464,Z 352.2,A -85,B 0,C 180,E1 -1519.836,E2 -1519.836} C_VEL
LIN {X 0,Y 587.366,Z 362.596,A -85,B 0,C 180,E1 -1520.617,E2 -1520.617} C_VEL
LIN {X 0,Y 587.322,Z 371.11,A -85,B 0,C 180,E1 -1521.397,E2 -1521.397} C_VEL
LIN {X 0,Y 587.274,Z 378.958,A -85,B 0,C 180,E1 -1522.263,E2 -1522.263} C_VEL
LIN {X 0,Y 587.23,Z 385.467,A -85,B 0,C 180,E1 -1523.126,E2 -1523.126} C_VEL
LIN {X 0,Y 587.237,Z 391.865,A -85,B 0,C 180,E1 -1524.161,E2 -1524.161} C_VEL
LIN {X 0,Y 587.147,Z 396.949,A -85,B 0,C 180,E1 -1525.193,E2 -1525.193} C_VEL
LIN {X 0,Y 587.213,Z 400.895,A -85,B 0,C 180,E1 -1526.225,E2 -1526.225} C_VEL
LIN {X 0,Y 587.132,Z 403.808,A -85,B 0,C 180,E1 -1527.255,E2 -1527.255} C_VEL
LIN {X 0,Y 587.141,Z 405.199,A -85,B 0,C 180,E1 -1527.942,E2 -1527.942} C_VEL
LIN {X 0,Y 587.14,Z 406.784,A -85,B 0,C 180,E1 -1529.314,E2 -1529.314} C_VEL
LIN {X 0,Y 587.137,Z 407,A -85,B 0,C 180,E1 -1530,E2 -1530} C_VEL
LIN {X 0,Y 587.147,Z 406.186,A -85,B 0,C 180,E1 -1531.371,E2 -1531.371} C_VEL
LIN {X 0,Y 587.141,Z 405.201,A -85,B 0,C 180,E1 -1532.058,E2 -1532.058} C_VEL
LIN {X 0,Y 587.132,Z 403.811,A -85,B 0,C 180,E1 -1532.744,E2 -1532.744} C_VEL
LIN {X 0,Y 587.213,Z 400.897,A -85,B 0,C 180,E1 -1533.774,E2 -1533.774} C_VEL
LIN {X 0,Y 587.147,Z 396.951,A -85,B 0,C 180,E1 -1534.806,E2 -1534.806} C_VEL
LIN {X 0,Y 587.218,Z 390.88,A -85,B 0,C 180,E1 -1536.011,E2 -1536.011} C_VEL
LIN {X 0,Y 587.244,Z 384.241,A -85,B 0,C 180,E1 -1537.046,E2 -1537.046} C_VEL
LIN {X 0,Y 587.299,Z 375.994,A -85,B 0,C 180,E1 -1538.083,E2 -1538.083} C_VEL
LIN {X 0,Y 587.343,Z 367.543,A -85,B 0,C 180,E1 -1538.948,E2 -1538.948} C_VEL
LIN {X 0,Y 587.419,Z 357.104,A -85,B 0,C 180,E1 -1539.816,E2 -1539.816} C_VEL
LIN {X 0,Y 587.497,Z 346.765,A -85,B 0,C 180,E1 -1540.511,E2 -1540.511} C_VEL
LIN {X 0,Y 587.56,Z 334.826,A -85,B 0,C 180,E1 -1541.148,E2 -1541.148} C_VEL
LIN {X 0,Y 587.628,Z 322.613,A -85,B 0,C 180,E1 -1541.639,E2 -1541.639} C_VEL
LIN {X 0,Y 587.703,Z 309.457,A -85,B 0,C 180,E1 -1542.013,E2 -1542.013} C_VEL
LIN {X 0,Y 587.784,Z 297.125,A -85,B 0,C 180,E1 -1542.231,E2 -1542.231} C_VEL
LIN {X 0,Y 587.708,Z 196.753,A -85,B 0,C 180,E1 -1543.465,E2 -1543.465} C_VEL
LIN {X 0,Y 587.381,Z 194.617,A -85,B 0,C 180,E1 -1543.514,E2 -1543.514} C_VEL
LIN {X 0,Y 587.541,Z 174.068,A -85,B 0,C 180,E1 -1546.325,E2 -1546.325} C_VEL
LIN {X 0,Y 587.668,Z 153.852,A -85,B 0,C 180,E1 -1549.13,E2 -1549.13} C_VEL
LIN {X 0,Y 587.822,Z 135.231,A -85,B 0,C 180,E1 -1551.754,E2 -1551.754} C_VEL
LIN {X 0,Y 587.607,Z 126.883,A -85,B 0,C 180,E1 -1552.934,E2 -1552.934} C_VEL
LIN {X 0,Y 587.313,Z 125.328,A -85,B 0,C 180,E1 -1553.179,E2 -1553.179} C_VEL
LIN {X 0,Y 587.328,Z 125.327,A -85,B 0,C 180,E1 -1555.516,E2 -1555.516} C_VEL
LIN {X 0,Y 587.299,Z 125.332,A -85,B 0,C 180,E1 -1557.819,E2 -1557.819} C_VEL
LIN {X 0,Y 587.315,Z 125.321,A -85,B 0,C 180,E1 -1560.506,E2 -1560.506} C_VEL
LIN {X 0,Y 587.322,Z 125.327,A -85,B 0,C 180,E1 -1563.396,E2 -1563.396} C_VEL
LIN {X 0,Y 587.274,Z 125.329,A -85,B 0,C 180,E1 -1565.9,E2 -1565.9} C_VEL
LIN {X 0,Y 587.307,Z 125.322,A -85,B 0,C 180,E1 -1568.48,E2 -1568.48} C_VEL
LIN {X 0,Y 587.329,Z 125.326,A -85,B 0,C 180,E1 -1571.156,E2 -1571.156} C_VEL
LIN {X 0,Y 587.306,Z 125.322,A -85,B 0,C 180,E1 -1574.111,E2 -1574.111} C_VEL
LIN {X 0,Y 587.285,Z 125.332,A -85,B 0,C 180,E1 -1576.991,E2 -1576.991} C_VEL
LIN {X 0,Y 587.295,Z 125.325,A -85,B 0,C 180,E1 -1579.744,E2 -1579.744} C_VEL
LIN {X 0,Y 587.33,Z 125.32,A -85,B 0,C 180,E1 -1582.391,E2 -1582.391} C_VEL
LIN {X 0,Y 587.319,Z 125.321,A -85,B 0,C 180,E1 -1585.655,E2 -1585.655} C_VEL
LIN {X 0,Y 587.322,Z 125.321,A -85,B 0,C 180,E1 -1588.23,E2 -1588.23} C_VEL
LIN {X 0,Y 587.328,Z 125.328,A -85,B 0,C 180,E1 -1590.868,E2 -1590.868} C_VEL
LIN {X 0,Y 587.302,Z 125.323,A -85,B 0,C 180,E1 -1593.828,E2 -1593.828} C_VEL
LIN {X 0,Y 587.283,Z 125.333,A -85,B 0,C 180,E1 -1596.74,E2 -1596.74} C_VEL
LIN {X 0,Y 587.302,Z 125.326,A -85,B 0,C 180,E1 -1598.967,E2 -1598.967} C_VEL
LIN {X 0,Y 587.309,Z 125.323,A -85,B 0,C 180,E1 -1601.15,E2 -1601.15} C_VEL
LIN {X 0,Y 587.276,Z 125.33,A -85,B 0,C 180,E1 -1604.023,E2 -1604.023} C_VEL
LIN {X 0,Y 587.321,Z 125.327,A -85,B 0,C 180,E1 -1606.153,E2 -1606.153} C_VEL
LIN {X 0,Y 587.306,Z 125.323,A -85,B 0,C 180,E1 -1608.962,E2 -1608.962} C_VEL
LIN {X 0,Y 587.315,Z 125.324,A -85,B 0,C 180,E1 -1611.744,E2 -1611.744} C_VEL
LIN {X 0,Y 587.321,Z 125.324,A -85,B 0,C 180,E1 -1614.507,E2 -1614.507} C_VEL
LIN {X 0,Y 587.321,Z 125.321,A -85,B 0,C 180,E1 -1617.257,E2 -1617.257} C_VEL
LIN {X 0,Y 587.37,Z 125.324,A -85,B 0,C 180,E1 -1620,E2 -1620} C_VEL
LIN {X 0,Y 587.324,Z 125.32,A -85,B 0,C 180,E1 -1622.744,E2 -1622.744} C_VEL
LIN {X 0,Y 587.33,Z 125.324,A -85,B 0,C 180,E1 -1625.493,E2 -1625.493} C_VEL
LIN {X 0,Y 587.321,Z 125.322,A -85,B 0,C 180,E1 -1628.256,E2 -1628.256} C_VEL
LIN {X 0,Y 587.319,Z 125.323,A -85,B 0,C 180,E1 -1631.125,E2 -1631.125} C_VEL
LIN {X 0,Y 587.307,Z 125.323,A -85,B 0,C 180,E1 -1634.242,E2 -1634.242} C_VEL
LIN {X 0,Y 587.269,Z 125.327,A -85,B 0,C 180,E1 -1636.792,E2 -1636.792} C_VEL
LIN {X 0,Y 587.27,Z 125.327,A -85,B 0,C 180,E1 -1638.27,E2 -1638.27} C_VEL
LIN {X 0,Y 586.633,Z 125.408,A -85,B 0,C 180,E1 -1638.842,E2 -1638.842} C_VEL
LIN {X 0,Y 583.832,Z 125.759,A -85,B 0,C 180,E1 -1639.771,E2 -1639.771} C_VEL
LIN {X 0,Y 581.435,Z 126.056,A -85,B 0,C 180,E1 -1640.518,E2 -1640.518} C_VEL
LIN {X 0,Y 580.376,Z 126.191,A -85,B 0,C 180,E1 -1641.095,E2 -1641.095} C_VEL
LIN {X 0,Y 580.275,Z 126.207,A -85,B 0,C 180,E1 -1641.29,E2 -1641.29} C_VEL
LIN {X 0,Y 580.24,Z 126.208,A -85,B 0,C 180,E1 -1643.56,E2 -1643.56} C_VEL
LIN {X 0,Y 580.254,Z 126.2,A -85,B 0,C 180,E1 -1646.329,E2 -1646.329} C_VEL
LIN {X 0,Y 580.264,Z 126.207,A -85,B 0,C 180,E1 -1649.305,E2 -1649.305} C_VEL
LIN {X 0,Y 580.275,Z 126.198,A -85,B 0,C 180,E1 -1652.202,E2 -1652.202} C_VEL
LIN {X 0,Y 580.276,Z 126.203,A -85,B 0,C 180,E1 -1654.697,E2 -1654.697} C_VEL
LIN {X 0,Y 580.288,Z 126.201,A -85,B 0,C 180,E1 -1657.269,E2 -1657.269} C_VEL
LIN {X 0,Y 580.276,Z 126.2,A -85,B 0,C 180,E1 -1660.27,E2 -1660.27} C_VEL
LIN {X 0,Y 580.25,Z 126.21,A -85,B 0,C 180,E1 -1662.709,E2 -1662.709} C_VEL
LIN {X 0,Y 580.25,Z 126.201,A -85,B 0,C 180,E1 -1665.612,E2 -1665.612} C_VEL
LIN {X 0,Y 580.269,Z 126.208,A -85,B 0,C 180,E1 -1668.671,E2 -1668.671} C_VEL
LIN {X 0,Y 580.264,Z 126.203,A -85,B 0,C 180,E1 -1670.965,E2 -1670.965} C_VEL
LIN {X 0,Y 580.243,Z 126.202,A -85,B 0,C 180,E1 -1673.596,E2 -1673.596} C_VEL
LIN {X 0,Y 580.297,Z 126.201,A -85,B 0,C 180,E1 -1676.145,E2 -1676.145} C_VEL
LIN {X 0,Y 580.265,Z 126.204,A -85,B 0,C 180,E1 -1678.615,E2 -1678.615} C_VEL
LIN {X 0,Y 580.281,Z 126.198,A -85,B 0,C 180,E1 -1681.024,E2 -1681.024} C_VEL
LIN {X 0,Y 580.266,Z 126.209,A -85,B 0,C 180,E1 -1684.151,E2 -1684.151} C_VEL
LIN {X 0,Y 580.257,Z 126.2,A -85,B 0,C 180,E1 -1687,E2 -1687} C_VEL
LIN {X 0,Y 580.265,Z 126.202,A -85,B 0,C 180,E1 -1689.438,E2 -1689.438} C_VEL
LIN {X 0,Y 580.316,Z 126.319,A -85,B 0,C 180,E1 -1691.029,E2 -1691.029} C_VEL
LIN {X 0,Y 580.438,Z 134.908,A -85,B 0,C 180,E1 -1692.581,E2 -1692.581} C_VEL
LIN {X 0,Y 580.374,Z 150.004,A -85,B 0,C 180,E1 -1695.269,E2 -1695.269} C_VEL
LIN {X 0,Y 580.331,Z 156.501,A -85,B 0,C 180,E1 -1696.402,E2 -1696.402} C_VEL
LIN {X 0,Y 580.957,Z 160.52,A -85,B 0,C 180,E1 -1696.468,E2 -1696.468} C_VEL
LIN {X 0,Y 580.808,Z 262.94,A -85,B 0,C 180,E1 -1697.753,E2 -1697.753} C_VEL
LIN {X 0,Y 580.72,Z 276.207,A -85,B 0,C 180,E1 -1698.061,E2 -1698.061} C_VEL
LIN {X 0,Y 580.65,Z 288.366,A -85,B 0,C 180,E1 -1698.481,E2 -1698.481} C_VEL
LIN {X 0,Y 580.554,Z 299.801,A -85,B 0,C 180,E1 -1699.009,E2 -1699.009} C_VEL
LIN {X 0,Y 580.447,Z 311.549,A -85,B 0,C 180,E1 -1699.713,E2 -1699.713} C_VEL
LIN {X 0,Y 580.346,Z 322.065,A -85,B 0,C 180,E1 -1700.503,E2 -1700.503} C_VEL
LIN {X 0,Y 580.272,Z 330.663,A -85,B 0,C 180,E1 -1701.293,E2 -1701.293} C_VEL
LIN {X 0,Y 580.222,Z 338.586,A -85,B 0,C 180,E1 -1702.169,E2 -1702.169} C_VEL
LIN {X 0,Y 580.168,Z 346.287,A -85,B 0,C 180,E1 -1703.21,E2 -1703.21} C_VEL
LIN {X 0,Y 580.139,Z 353.448,A -85,B 0,C 180,E1 -1704.439,E2 -1704.439} C_VEL
LIN {X 0,Y 580.108,Z 358.19,A -85,B 0,C 180,E1 -1705.484,E2 -1705.484} C_VEL
LIN {X 0,Y 580.123,Z 361.823,A -85,B 0,C 180,E1 -1706.528,E2 -1706.528} C_VEL
LIN {X 0,Y 580.043,Z 363.7,A -85,B 0,C 180,E1 -1707.222,E2 -1707.222} C_VEL
LIN {X 0,Y 580.04,Z 365.127,A -85,B 0,C 180,E1 -1707.917,E2 -1707.917} C_VEL
LIN {X 0,Y 580.04,Z 366.755,A -85,B 0,C 180,E1 -1709.306,E2 -1709.306} C_VEL
LIN {X 0,Y 580.038,Z 366.996,A -85,B 0,C 180,E1 -1710,E2 -1710} C_VEL
LIN {X 0,Y 580.04,Z 366.815,A -85,B 0,C 180,E1 -1710.695,E2 -1710.695} C_VEL
LIN {X 0,Y 580.04,Z 365.27,A -85,B 0,C 180,E1 -1712.083,E2 -1712.083} C_VEL
LIN {X 0,Y 580.044,Z 363.909,A -85,B 0,C 180,E1 -1712.778,E2 -1712.778} C_VEL
LIN {X 0,Y 580.11,Z 361.033,A -85,B 0,C 180,E1 -1713.821,E2 -1713.821} C_VEL
LIN {X 0,Y 580.053,Z 357.132,A -85,B 0,C 180,E1 -1714.866,E2 -1714.866} C_VEL
LIN {X 0,Y 580.163,Z 352.101,A -85,B 0,C 180,E1 -1715.91,E2 -1715.91} C_VEL
LIN {X 0,Y 580.158,Z 345.778,A -85,B 0,C 180,E1 -1716.958,E2 -1716.958} C_VEL
LIN {X 0,Y 580.241,Z 337.857,A -85,B 0,C 180,E1 -1718.007,E2 -1718.007} C_VEL
LIN {X 0,Y 580.308,Z 328.008,A -85,B 0,C 180,E1 -1719.059,E2 -1719.059} C_VEL
LIN {X 0,Y 580.418,Z 317.69,A -85,B 0,C 180,E1 -1719.936,E2 -1719.936} C_VEL
LIN {X 0,Y 580.493,Z 306.05,A -85,B 0,C 180,E1 -1720.728,E2 -1720.728} C_VEL
LIN {X 0,Y 580.621,Z 294.4,A -85,B 0,C 180,E1 -1721.348,E2 -1721.348} C_VEL
LIN {X 0,Y 580.666,Z 282.621,A -85,B 0,C 180,E1 -1721.825,E2 -1721.825} C_VEL
LIN {X 0,Y 580.769,Z 269.457,A -85,B 0,C 180,E1 -1722.204,E2 -1722.204} C_VEL
LIN {X 0,Y 580.853,Z 257.117,A -85,B 0,C 180,E1 -1722.424,E2 -1722.424} C_VEL
LIN {X 0,Y 580.872,Z 160.082,A -85,B 0,C 180,E1 -1723.63,E2 -1723.63} C_VEL
LIN {X 0,Y 580.31,Z 156.336,A -85,B 0,C 180,E1 -1723.705,E2 -1723.705} C_VEL
LIN {X 0,Y 580.427,Z 140.372,A -85,B 0,C 180,E1 -1726.532,E2 -1726.532} C_VEL
LIN {X 0,Y 580.418,Z 127.196,A -85,B 0,C 180,E1 -1728.899,E2 -1728.899} C_VEL
LIN {X 0,Y 580.298,Z 126.2,A -85,B 0,C 180,E1 -1729.087,E2 -1729.087} C_VEL
LIN {X 0,Y 580.258,Z 126.21,A -85,B 0,C 180,E1 -1732.053,E2 -1732.053} C_VEL
LIN {X 0,Y 580.29,Z 126.196,A -85,B 0,C 180,E1 -1735.081,E2 -1735.081} C_VEL
LIN {X 0,Y 580.277,Z 126.202,A -85,B 0,C 180,E1 -1738.187,E2 -1738.187} C_VEL
LIN {X 0,Y 580.272,Z 126.198,A -85,B 0,C 180,E1 -1740.692,E2 -1740.692} C_VEL
LIN {X 0,Y 580.302,Z 126.198,A -85,B 0,C 180,E1 -1743.316,E2 -1743.316} C_VEL
LIN {X 0,Y 580.243,Z 126.21,A -85,B 0,C 180,E1 -1745.755,E2 -1745.755} C_VEL
LIN {X 0,Y 580.282,Z 126.199,A -85,B 0,C 180,E1 -1748.147,E2 -1748.147} C_VEL
LIN {X 0,Y 580.296,Z 126.197,A -85,B 0,C 180,E1 -1750.843,E2 -1750.843} C_VEL
LIN {X 0,Y 580.269,Z 126.204,A -85,B 0,C 180,E1 -1753.659,E2 -1753.659} C_VEL
LIN {X 0,Y 580.242,Z 126.203,A -85,B 0,C 180,E1 -1756.613,E2 -1756.613} C_VEL
LIN {X 0,Y 580.292,Z 126.204,A -85,B 0,C 180,E1 -1759.156,E2 -1759.156} C_VEL
LIN {X 0,Y 580.281,Z 126.198,A -85,B 0,C 180,E1 -1761.928,E2 -1761.928} C_VEL
LIN {X 0,Y 580.229,Z 126.205,A -85,B 0,C 180,E1 -1764.451,E2 -1764.451} C_VEL
LIN {X 0,Y 580.281,Z 126.207,A -85,B 0,C 180,E1 -1766.974,E2 -1766.974} C_VEL
LIN {X 0,Y 580.268,Z 126.202,A -85,B 0,C 180,E1 -1769.423,E2 -1769.423} C_VEL
LIN {X 0,Y 580.241,Z 126.203,A -85,B 0,C 180,E1 -1772.151,E2 -1772.151} C_VEL
LIN {X 0,Y 580.276,Z 126.206,A -85,B 0,C 180,E1 -1774.919,E2 -1774.919} C_VEL
LIN {X 0,Y 580.249,Z 126.202,A -85,B 0,C 180,E1 -1777.946,E2 -1777.946} C_VEL
LIN {X 0,Y 580.293,Z 126.202,A -85,B 0,C 180,E1 -1780.849,E2 -1780.849} C_VEL
LIN {X 0,Y 580.232,Z 126.204,A -85,B 0,C 180,E1 -1783.824,E2 -1783.824} C_VEL
LIN {X 0,Y 580.288,Z 126.199,A -85,B 0,C 180,E1 -1785.982,E2 -1785.982} C_VEL
LIN {X 0,Y 580.302,Z 126.198,A -85,B 0,C 180,E1 -1788.827,E2 -1788.827} C_VEL
LIN {X 0,Y 580.294,Z 126.196,A -85,B 0,C 180,E1 -1791.643,E2 -1791.643} C_VEL
LIN {X 0,Y 580.298,Z 126.202,A -85,B 0,C 180,E1 -1794.44,E2 -1794.44} C_VEL
LIN {X 0,Y 580.335,Z 126.197,A -85,B 0,C 180,E1 -1797.918,E2 -1797.918} C_VEL
LIN {X 0,Y 580.344,Z 126.198,A -85,B 0,C 180,E1 -1800,E2 -1800} C_VEL
LIN {X 0,Y 580.296,Z 126.196,A -85,B 0,C 180,E1 -1802.777,E2 -1802.777} C_VEL
LIN {X 0,Y 580.292,Z 126.2,A -85,B 0,C 180,E1 -1805.56,E2 -1805.56} C_VEL
LIN {X 0,Y 580.285,Z 126.199,A -85,B 0,C 180,E1 -1808.357,E2 -1808.357} C_VEL
LIN {X 0,Y 580.263,Z 126.201,A -85,B 0,C 180,E1 -1811.174,E2 -1811.174} C_VEL
LIN {X 0,Y 580.274,Z 126.199,A -85,B 0,C 180,E1 -1814.324,E2 -1814.324} C_VEL
LIN {X 0,Y 580.246,Z 126.202,A -85,B 0,C 180,E1 -1816.899,E2 -1816.899} C_VEL
LIN {X 0,Y 580.263,Z 126.204,A -85,B 0,C 180,E1 -1819.824,E2 -1819.824} C_VEL
LIN {X 0,Y 580.223,Z 126.206,A -85,B 0,C 180,E1 -1822.055,E2 -1822.055} C_VEL
LIN {X 0,Y 580.245,Z 126.203,A -85,B 0,C 180,E1 -1824.715,E2 -1824.715} C_VEL
LIN {X 0,Y 580.244,Z 126.21,A -85,B 0,C 180,E1 -1827.404,E2 -1827.404} C_VEL
LIN {X 0,Y 580.242,Z 126.204,A -85,B 0,C 180,E1 -1829.775,E2 -1829.775} C_VEL
LIN {X 0,Y 580.279,Z 126.197,A -85,B 0,C 180,E1 -1832.202,E2 -1832.202} C_VEL
LIN {X 0,Y 580.269,Z 126.202,A -85,B 0,C 180,E1 -1834.698,E2 -1834.698} C_VEL
LIN {X 0,Y 580.282,Z 126.203,A -85,B 0,C 180,E1 -1837.27,E2 -1837.27} C_VEL
LIN {X 0,Y 580.279,Z 126.199,A -85,B 0,C 180,E1 -1840.269,E2 -1840.269} C_VEL
LIN {X 0,Y 580.251,Z 126.208,A -85,B 0,C 180,E1 -1842.709,E2 -1842.709} C_VEL
LIN {X 0,Y 580.249,Z 126.201,A -85,B 0,C 180,E1 -1845.611,E2 -1845.611} C_VEL
LIN {X 0,Y 580.267,Z 126.209,A -85,B 0,C 180,E1 -1848.671,E2 -1848.671} C_VEL
LIN {X 0,Y 580.261,Z 126.204,A -85,B 0,C 180,E1 -1850.964,E2 -1850.964} C_VEL
LIN {X 0,Y 580.243,Z 126.202,A -85,B 0,C 180,E1 -1853.595,E2 -1853.595} C_VEL
LIN {X 0,Y 580.273,Z 126.203,A -85,B 0,C 180,E1 -1856.143,E2 -1856.143} C_VEL
LIN {X 0,Y 580.267,Z 126.206,A -85,B 0,C 180,E1 -1858.614,E2 -1858.614} C_VEL
LIN {X 0,Y 580.282,Z 126.199,A -85,B 0,C 180,E1 -1861.023,E2 -1861.023} C_VEL
LIN {X 0,Y 580.265,Z 126.209,A -85,B 0,C 180,E1 -1864.15,E2 -1864.15} C_VEL
LIN {X 0,Y 580.29,Z 126.323,A -85,B 0,C 180,E1 -1866.717,E2 -1866.717} C_VEL
LIN {X 0,Y 580.899,Z 131.021,A -85,B 0,C 180,E1 -1867.41,E2 -1867.41} C_VEL
LIN {X 0,Y 580.779,Z 151.92,A -85,B 0,C 180,E1 -1870.359,E2 -1870.359} C_VEL
LIN {X 0,Y 580.562,Z 174.062,A -85,B 0,C 180,E1 -1873.472,E2 -1873.472} C_VEL
LIN {X 0,Y 580.384,Z 194.612,A -85,B 0,C 180,E1 -1876.319,E2 -1876.319} C_VEL
LIN {X 0,Y 580.936,Z 200.495,A -85,B 0,C 180,E1 -1876.422,E2 -1876.422} C_VEL
LIN {X 0,Y 580.806,Z 302.937,A -85,B 0,C 180,E1 -1877.708,E2 -1877.708} C_VEL
LIN {X 0,Y 580.727,Z 316.212,A -85,B 0,C 180,E1 -1878.017,E2 -1878.017} C_VEL
LIN {X 0,Y 580.648,Z 328.37,A -85,B 0,C 180,E1 -1878.436,E2 -1878.436} C_VEL
LIN {X 0,Y 580.579,Z 340.624,A -85,B 0,C 180,E1 -1879.009,E2 -1879.009} C_VEL
LIN {X 0,Y 580.441,Z 352.198,A -85,B 0,C 180,E1 -1879.712,E2 -1879.712} C_VEL
LIN {X 0,Y 580.345,Z 362.598,A -85,B 0,C 180,E1 -1880.503,E2 -1880.503} C_VEL
LIN {X 0,Y 580.271,Z 371.11,A -85,B 0,C 180,E1 -1881.292,E2 -1881.292} C_VEL
LIN {X 0,Y 580.222,Z 378.958,A -85,B 0,C 180,E1 -1882.168,E2 -1882.168} C_VEL
LIN {X 0,Y 580.154,Z 386.65,A -85,B 0,C 180,E1 -1883.221,E2 -1883.221} C_VEL
LIN {X 0,Y 580.139,Z 393.678,A -85,B 0,C 180,E1 -1884.438,E2 -1884.438} C_VEL
LIN {X 0,Y 580.108,Z 398.371,A -85,B 0,C 180,E1 -1885.483,E2 -1885.483} C_VEL
LIN {X 0,Y 580.123,Z 401.956,A -85,B 0,C 180,E1 -1886.527,E2 -1886.527} C_VEL
LIN {X 0,Y 580.043,Z 403.807,A -85,B 0,C 180,E1 -1887.222,E2 -1887.222} C_VEL
LIN {X 0,Y 580.04,Z 405.198,A -85,B 0,C 180,E1 -1887.917,E2 -1887.917} C_VEL
LIN {X 0,Y 580.04,Z 406.785,A -85,B 0,C 180,E1 -1889.305,E2 -1889.305} C_VEL
LIN {X 0,Y 580.037,Z 407,A -85,B 0,C 180,E1 -1890,E2 -1890} C_VEL
LIN {X 0,Y 580.047,Z 406.187,A -85,B 0,C 180,E1 -1891.388,E2 -1891.388} C_VEL
LIN {X 0,Y 580.04,Z 405.2,A -85,B 0,C 180,E1 -1892.083,E2 -1892.083} C_VEL
LIN {X 0,Y 580.043,Z 403.811,A -85,B 0,C 180,E1 -1892.778,E2 -1892.778} C_VEL
LIN {X 0,Y 580.11,Z 400.897,A -85,B 0,C 180,E1 -1893.82,E2 -1893.82} C_VEL
LIN {X 0,Y 580.053,Z 396.951,A -85,B 0,C 180,E1 -1894.865,E2 -1894.865} C_VEL
LIN {X 0,Y 580.139,Z 390.879,A -85,B 0,C 180,E1 -1896.084,E2 -1896.084} C_VEL
LIN {X 0,Y 580.184,Z 384.241,A -85,B 0,C 180,E1 -1897.132,E2 -1897.132} C_VEL
LIN {X 0,Y 580.25,Z 375.995,A -85,B 0,C 180,E1 -1898.181,E2 -1898.181} C_VEL
LIN {X 0,Y 580.308,Z 367.544,A -85,B 0,C 180,E1 -1899.058,E2 -1899.058} C_VEL
LIN {X 0,Y 580.422,Z 357.105,A -85,B 0,C 180,E1 -1899.935,E2 -1899.935} C_VEL
LIN {X 0,Y 580.506,Z 346.763,A -85,B 0,C 180,E1 -1900.639,E2 -1900.639} C_VEL
LIN {X 0,Y 580.595,Z 335.255,A -85,B 0,C 180,E1 -1901.263,E2 -1901.263} C_VEL
LIN {X 0,Y 580.682,Z 322.488,A -85,B 0,C 180,E1 -1901.784,E2 -1901.784} C_VEL
LIN {X 0,Y 580.777,Z 309.456,A -85,B 0,C 180,E1 -1902.159,E2 -1902.159} C_VEL
LIN {X 0,Y 580.858,Z 297.125,A -85,B 0,C 180,E1 -1902.379,E2 -1902.379} C_VEL
LIN {X 0,Y 580.793,Z 197.426,A -85,B 0,C 180,E1 -1903.62,E2 -1903.62} C_VEL
LIN {X 0,Y 580.386,Z 194.617,A -85,B 0,C 180,E1 -1903.68,E2 -1903.68} C_VEL
LIN {X 0,Y 580.566,Z 172.773,A -85,B 0,C 180,E1 -1906.708,E2 -1906.708} C_VEL
LIN {X 0,Y 580.782,Z 150.768,A -85,B 0,C 180,E1 -1909.805,E2 -1909.805} C_VEL
LIN {X 0,Y 580.894,Z 131.026,A -85,B 0,C 180,E1 -1912.589,E2 -1912.589} C_VEL
LIN {X 0,Y 580.275,Z 126.206,A -85,B 0,C 180,E1 -1913.301,E2 -1913.301} C_VEL
LIN {X 0,Y 580.264,Z 126.209,A -85,B 0,C 180,E1 -1915.85,E2 -1915.85} C_VEL
LIN {X 0,Y 580.28,Z 126.199,A -85,B 0,C 180,E1 -1918.976,E2 -1918.976} C_VEL
LIN {X 0,Y 580.264,Z 126.206,A -85,B 0,C 180,E1 -1921.385,E2 -1921.385} C_VEL
LIN {X 0,Y 580.272,Z 126.203,A -85,B 0,C 180,E1 -1923.857,E2 -1923.857} C_VEL
LIN {X 0,Y 580.272,Z 126.201,A -85,B 0,C 180,E1 -1926.93,E2 -1926.93} C_VEL
LIN {X 0,Y 580.269,Z 126.2,A -85,B 0,C 180,E1 -1929.934,E2 -1929.934} C_VEL
LIN {X 0,Y 580.252,Z 126.202,A -85,B 0,C 180,E1 -1932.707,E2 -1932.707} C_VEL
LIN {X 0,Y 580.244,Z 126.205,A -85,B 0,C 180,E1 -1935.61,E2 -1935.61} C_VEL
LIN {X 0,Y 580.263,Z 126.202,A -85,B 0,C 180,E1 -1938.669,E2 -1938.669} C_VEL
LIN {X 0,Y 580.26,Z 126.208,A -85,B 0,C 180,E1 -1940.963,E2 -1940.963} C_VEL
LIN {X 0,Y 580.236,Z 126.204,A -85,B 0,C 180,E1 -1943.594,E2 -1943.594} C_VEL
LIN {X 0,Y 580.262,Z 126.2,A -85,B 0,C 180,E1 -1946.142,E2 -1946.142} C_VEL
LIN {X 0,Y 580.256,Z 126.206,A -85,B 0,C 180,E1 -1948.613,E2 -1948.613} C_VEL
LIN {X 0,Y 580.266,Z 126.205,A -85,B 0,C 180,E1 -1951.022,E2 -1951.022} C_VEL
LIN {X 0,Y 580.258,Z 126.2,A -85,B 0,C 180,E1 -1953.67,E2 -1953.67} C_VEL
LIN {X 0,Y 580.235,Z 126.21,A -85,B 0,C 180,E1 -1956.44,E2 -1956.44} C_VEL
LIN {X 0,Y 580.239,Z 126.202,A -85,B 0,C 180,E1 -1959.436,E2 -1959.436} C_VEL
LIN {X 0,Y 580.223,Z 126.205,A -85,B 0,C 180,E1 -1961.644,E2 -1961.644} C_VEL
LIN {X 0,Y 580.254,Z 126.208,A -85,B 0,C 180,E1 -1964.546,E2 -1964.546} C_VEL
LIN {X 0,Y 580.221,Z 126.209,A -85,B 0,C 180,E1 -1966.695,E2 -1966.695} C_VEL
LIN {X 0,Y 580.255,Z 126.202,A -85,B 0,C 180,E1 -1968.826,E2 -1968.826} C_VEL
LIN {X 0,Y 580.281,Z 126.199,A -85,B 0,C 180,E1 -1971.643,E2 -1971.643} C_VEL
LIN {X 0,Y 580.29,Z 126.201,A -85,B 0,C 180,E1 -1974.44,E2 -1974.44} C_VEL
LIN {X 0,Y 580.332,Z 126.199,A -85,B 0,C 180,E1 -1977.918,E2 -1977.918} C_VEL
LIN {X 0,Y 580.338,Z 126.2,A -85,B 0,C 180,E1 -1980,E2 -1980} C_VEL
LIN {X 0,Y 580.292,Z 126.196,A -85,B 0,C 180,E1 -1982.777,E2 -1982.777} C_VEL
LIN {X 0,Y 580.299,Z 126.201,A -85,B 0,C 180,E1 -1985.56,E2 -1985.56} C_VEL
LIN {X 0,Y 580.289,Z 126.197,A -85,B 0,C 180,E1 -1988.357,E2 -1988.357} C_VEL
LIN {X 0,Y 580.29,Z 126.199,A -85,B 0,C 180,E1 -1991.191,E2 -1991.191} C_VEL
LIN {X 0,Y 580.283,Z 126.2,A -85,B 0,C 180,E1 -1994.018,E2 -1994.018} C_VEL
LIN {X 0,Y 580.218,Z 126.207,A -85,B 0,C 180,E1 -1996.9,E2 -1996.9} C_VEL
LIN {X 0,Y 580.264,Z 126.203,A -85,B 0,C 180,E1 -1999.824,E2 -1999.824} C_VEL
LIN {X 0,Y 580.275,Z 126.207,A -85,B 0,C 180,E1 -2001.29,E2 -2001.29} C_VEL
LIN {X 0,Y 579.562,Z 126.302,A -85,B 0,C 180,E1 -2001.869,E2 -2001.869} C_VEL
LIN {X 0,Y 576.675,Z 126.658,A -85,B 0,C 180,E1 -2002.809,E2 -2002.809} C_VEL
LIN {X 0,Y 574.273,Z 126.951,A -85,B 0,C 180,E1 -2003.565,E2 -2003.565} C_VEL
LIN {X 0,Y 573.26,Z 127.072,A -85,B 0,C 180,E1 -2004.149,E2 -2004.149} C_VEL
LIN {X 0,Y 573.187,Z 127.081,A -85,B 0,C 180,E1 -2004.347,E2 -2004.347} C_VEL
LIN {X 0,Y 573.191,Z 127.086,A -85,B 0,C 180,E1 -2006.979,E2 -2006.979} C_VEL
LIN {X 0,Y 573.21,Z 127.082,A -85,B 0,C 180,E1 -2009.484,E2 -2009.484} C_VEL
LIN {X 0,Y 573.228,Z 127.076,A -85,B 0,C 180,E1 -2012.226,E2 -2012.226} C_VEL
LIN {X 0,Y 573.223,Z 127.082,A -85,B 0,C 180,E1 -2014.771,E2 -2014.771} C_VEL
LIN {X 0,Y 573.223,Z 127.076,A -85,B 0,C 180,E1 -2017.809,E2 -2017.809} C_VEL
LIN {X 0,Y 573.239,Z 127.079,A -85,B 0,C 180,E1 -2020.526,E2 -2020.526} C_VEL
LIN {X 0,Y 573.2,Z 127.079,A -85,B 0,C 180,E1 -2023.666,E2 -2023.666} C_VEL
LIN {X 0,Y 573.225,Z 127.086,A -85,B 0,C 180,E1 -2026.641,E2 -2026.641} C_VEL
LIN {X 0,Y 573.241,Z 127.074,A -85,B 0,C 180,E1 -2029.476,E2 -2029.476} C_VEL
LIN {X 0,Y 573.224,Z 127.081,A -85,B 0,C 180,E1 -2032.193,E2 -2032.193} C_VEL
LIN {X 0,Y 573.228,Z 127.076,A -85,B 0,C 180,E1 -2035.23,E2 -2035.23} C_VEL
LIN {X 0,Y 573.243,Z 127.075,A -85,B 0,C 180,E1 -2037.774,E2 -2037.774} C_VEL
LIN {X 0,Y 573.238,Z 127.079,A -85,B 0,C 180,E1 -2040.634,E2 -2040.634} C_VEL
LIN {X 0,Y 573.212,Z 127.079,A -85,B 0,C 180,E1 -2043.513,E2 -2043.513} C_VEL
LIN {X 0,Y 573.212,Z 127.088,A -85,B 0,C 180,E1 -2046.134,E2 -2046.134} C_VEL
LIN {X 0,Y 573.246,Z 127.075,A -85,B 0,C 180,E1 -2049.174,E2 -2049.174} C_VEL
LIN {X 0,Y 573.28,Z 127.105,A -85,B 0,C 180,E1 -2050.943,E2 -2050.943} C_VEL
LIN {X 0,Y 573.432,Z 135.825,A -85,B 0,C 180,E1 -2052.527,E2 -2052.527} C_VEL
LIN {X 0,Y 573.329,Z 150.007,A -85,B 0,C 180,E1 -2055.083,E2 -2055.083} C_VEL
LIN {X 0,Y 573.31,Z 156.547,A -85,B 0,C 180,E1 -2056.233,E2 -2056.233} C_VEL
LIN {X 0,Y 574.04,Z 162.353,A -85,B 0,C 180,E1 -2056.324,E2 -2056.324} C_VEL
LIN {X 0,Y 573.875,Z 262.969,A -85,B 0,C 180,E1 -2057.603,E2 -2057.603} C_VEL
LIN {X 0,Y 573.784,Z 276.224,A -85,B 0,C 180,E1 -2057.915,E2 -2057.915} C_VEL
LIN {X 0,Y 573.707,Z 288.381,A -85,B 0,C 180,E1 -2058.34,E2 -2058.34} C_VEL
LIN {X 0,Y 573.583,Z 299.908,A -85,B 0,C 180,E1 -2058.879,E2 -2058.879} C_VEL
LIN {X 0,Y 573.432,Z 311.555,A -85,B 0,C 180,E1 -2059.586,E2 -2059.586} C_VEL
LIN {X 0,Y 573.333,Z 322.073,A -85,B 0,C 180,E1 -2060.386,E2 -2060.386} C_VEL
LIN {X 0,Y 573.241,Z 330.669,A -85,B 0,C 180,E1 -2061.185,E2 -2061.185} C_VEL
LIN {X 0,Y 573.161,Z 338.59,A -85,B 0,C 180,E1 -2062.072,E2 -2062.072} C_VEL
LIN {X 0,Y 573.092,Z 346.527,A -85,B 0,C 180,E1 -2063.163,E2 -2063.163} C_VEL
LIN {X 0,Y 573.071,Z 353.451,A -85,B 0,C 180,E1 -2064.37,E2 -2064.37} C_VEL
LIN {X 0,Y 573.028,Z 358.192,A -85,B 0,C 180,E1 -2065.428,E2 -2065.428} C_VEL
LIN {X 0,Y 573.022,Z 361.826,A -85,B 0,C 180,E1 -2066.485,E2 -2066.485} C_VEL
LIN {X 0,Y 572.959,Z 363.702,A -85,B 0,C 180,E1 -2067.188,E2 -2067.188} C_VEL
LIN {X 0,Y 572.94,Z 365.127,A -85,B 0,C 180,E1 -2067.891,E2 -2067.891} C_VEL
LIN {X 0,Y 572.941,Z 366.756,A -85,B 0,C 180,E1 -2069.298,E2 -2069.298} C_VEL
LIN {X 0,Y 572.939,Z 366.996,A -85,B 0,C 180,E1 -2070,E2 -2070} C_VEL
LIN {X 0,Y 572.94,Z 366.815,A -85,B 0,C 180,E1 -2070.703,E2 -2070.703} C_VEL
LIN {X 0,Y 572.94,Z 365.268,A -85,B 0,C 180,E1 -2072.109,E2 -2072.109} C_VEL
LIN {X 0,Y 572.96,Z 363.907,A -85,B 0,C 180,E1 -2072.813,E2 -2072.813} C_VEL
LIN {X 0,Y 573.015,Z 361.03,A -85,B 0,C 180,E1 -2073.868,E2 -2073.868} C_VEL
LIN {X 0,Y 572.963,Z 357.13,A -85,B 0,C 180,E1 -2074.926,E2 -2074.926} C_VEL
LIN {X 0,Y 573.076,Z 352.098,A -85,B 0,C 180,E1 -2075.984,E2 -2075.984} C_VEL
LIN {X 0,Y 573.083,Z 345.774,A -85,B 0,C 180,E1 -2077.044,E2 -2077.044} C_VEL
LIN {X 0,Y 573.175,Z 337.852,A -85,B 0,C 180,E1 -2078.106,E2 -2078.106} C_VEL
LIN {X 0,Y 573.287,Z 328.001,A -85,B 0,C 180,E1 -2079.17,E2 -2079.17} C_VEL
LIN {X 0,Y 573.421,Z 317.685,A -85,B 0,C 180,E1 -2080.059,E2 -2080.059} C_VEL
LIN {X 0,Y 573.49,Z 306.127,A -85,B 0,C 180,E1 -2080.855,E2 -2080.855} C_VEL
LIN {X 0,Y 573.658,Z 295.195,A -85,B 0,C 180,E1 -2081.449,E2 -2081.449} C_VEL
LIN {X 0,Y 573.731,Z 282.605,A -85,B 0,C 180,E1 -2081.97,E2 -2081.97} C_VEL
LIN {X 0,Y 573.844,Z 269.433,A -85,B 0,C 180,E1 -2082.354,E2 -2082.354} C_VEL
LIN {X 0,Y 573.943,Z 257.076,A -85,B 0,C 180,E1 -2082.576,E2 -2082.576} C_VEL
LIN {X 0,Y 573.93,Z 160.381,A -85,B 0,C 180,E1 -2083.794,E2 -2083.794} C_VEL
LIN {X 0,Y 573.267,Z 156.332,A -85,B 0,C 180,E1 -2083.877,E2 -2083.877} C_VEL
LIN {X 0,Y 573.398,Z 140.52,A -85,B 0,C 180,E1 -2086.713,E2 -2086.713} C_VEL
LIN {X 0,Y 573.433,Z 128.322,A -85,B 0,C 180,E1 -2088.922,E2 -2088.922} C_VEL
LIN {X 0,Y 573.254,Z 127.078,A -85,B 0,C 180,E1 -2089.173,E2 -2089.173} C_VEL
LIN {X 0,Y 573.226,Z 127.081,A -85,B 0,C 180,E1 -2091.581,E2 -2091.581} C_VEL
LIN {X 0,Y 573.216,Z 127.086,A -85,B 0,C 180,E1 -2093.866,E2 -2093.866} C_VEL
LIN {X 0,Y 573.215,Z 127.079,A -85,B 0,C 180,E1 -2096.487,E2 -2096.487} C_VEL
LIN {X 0,Y 573.243,Z 127.077,A -85,B 0,C 180,E1 -2099.367,E2 -2099.367} C_VEL
LIN {X 0,Y 573.248,Z 127.076,A -85,B 0,C 180,E1 -2102.227,E2 -2102.227} C_VEL
LIN {X 0,Y 573.232,Z 127.075,A -85,B 0,C 180,E1 -2104.77,E2 -2104.77} C_VEL
LIN {X 0,Y 573.228,Z 127.082,A -85,B 0,C 180,E1 -2107.808,E2 -2107.808} C_VEL
LIN {X 0,Y 573.246,Z 127.073,A -85,B 0,C 180,E1 -2110.525,E2 -2110.525} C_VEL
LIN {X 0,Y 573.235,Z 127.08,A -85,B 0,C 180,E1 -2113.668,E2 -2113.668} C_VEL
LIN {X 0,Y 573.207,Z 127.079,A -85,B 0,C 180,E1 -2116.638,E2 -2116.638} C_VEL
LIN {X 0,Y 573.244,Z 127.08,A -85,B 0,C 180,E1 -2119.475,E2 -2119.475} C_VEL
LIN {X 0,Y 573.225,Z 127.076,A -85,B 0,C 180,E1 -2122.191,E2 -2122.191} C_VEL
LIN {X 0,Y 573.222,Z 127.084,A -85,B 0,C 180,E1 -2125.23,E2 -2125.23} C_VEL
LIN {X 0,Y 573.234,Z 127.075,A -85,B 0,C 180,E1 -2127.774,E2 -2127.774} C_VEL
LIN {X 0,Y 573.229,Z 127.081,A -85,B 0,C 180,E1 -2130.632,E2 -2130.632} C_VEL
LIN {X 0,Y 573.227,Z 127.077,A -85,B 0,C 180,E1 -2133.509,E2 -2133.509} C_VEL
LIN {X 0,Y 573.193,Z 127.081,A -85,B 0,C 180,E1 -2136.133,E2 -2136.133} C_VEL
LIN {X 0,Y 573.248,Z 127.083,A -85,B 0,C 180,E1 -2138.709,E2 -2138.709} C_VEL
LIN {X 0,Y 573.192,Z 127.081,A -85,B 0,C 180,E1 -2141.41,E2 -2141.41} C_VEL
LIN {X 0,Y 573.201,Z 127.086,A -85,B 0,C 180,E1 -2144.351,E2 -2144.351} C_VEL
LIN {X 0,Y 573.192,Z 127.089,A -85,B 0,C 180,E1 -2146.528,E2 -2146.528} C_VEL
LIN {X 0,Y 573.253,Z 127.073,A -85,B 0,C 180,E1 -2149.403,E2 -2149.403} C_VEL
LIN {X 0,Y 573.216,Z 127.086,A -85,B 0,C 180,E1 -2152.249,E2 -2152.249} C_VEL
LIN {X 0,Y 573.269,Z 127.071,A -85,B 0,C 180,E1 -2155.077,E2 -2155.077} C_VEL
LIN {X 0,Y 573.305,Z 127.072,A -85,B 0,C 180,E1 -2157.892,E2 -2157.892} C_VEL
LIN {X 0,Y 573.312,Z 127.074,A -85,B 0,C 180,E1 -2160,E2 -2160} C_VEL
LIN {X 0,Y 573.264,Z 127.072,A -85,B 0,C 180,E1 -2162.811,E2 -2162.811} C_VEL
LIN {X 0,Y 573.26,Z 127.077,A -85,B 0,C 180,E1 -2165.628,E2 -2165.628} C_VEL
LIN {X 0,Y 573.226,Z 127.077,A -85,B 0,C 180,E1 -2168.46,E2 -2168.46} C_VEL
LIN {X 0,Y 573.23,Z 127.079,A -85,B 0,C 180,E1 -2171.313,E2 -2171.313} C_VEL
LIN {X 0,Y 573.23,Z 127.076,A -85,B 0,C 180,E1 -2174.406,E2 -2174.406} C_VEL
LIN {X 0,Y 573.186,Z 127.084,A -85,B 0,C 180,E1 -2177.114,E2 -2177.114} C_VEL
LIN {X 0,Y 573.197,Z 127.081,A -85,B 0,C 180,E1 -2180.079,E2 -2180.079} C_VEL
LIN {X 0,Y 573.189,Z 127.081,A -85,B 0,C 180,E1 -2182.34,E2 -2182.34} C_VEL
LIN {X 0,Y 573.205,Z 127.088,A -85,B 0,C 180,E1 -2185.412,E2 -2185.412} C_VEL
LIN {X 0,Y 573.19,Z 127.081,A -85,B 0,C 180,E1 -2188.018,E2 -2188.018} C_VEL
LIN {X 0,Y 573.2,Z 127.084,A -85,B 0,C 180,E1 -2190.878,E2 -2190.878} C_VEL
LIN {X 0,Y 573.239,Z 127.078,A -85,B 0,C 180,E1 -2193.521,E2 -2193.521} C_VEL
LIN {X 0,Y 573.183,Z 127.081,A -85,B 0,C 180,E1 -2196.054,E2 -2196.054} C_VEL
LIN {X 0,Y 573.23,Z 127.081,A -85,B 0,C 180,E1 -2198.703,E2 -2198.703} C_VEL
LIN {X 0,Y 573.205,Z 127.079,A -85,B 0,C 180,E1 -2201.59,E2 -2201.59} C_VEL
LIN {X 0,Y 573.206,Z 127.086,A -85,B 0,C 180,E1 -2204.673,E2 -2204.673} C_VEL
LIN {X 0,Y 573.209,Z 127.078,A -85,B 0,C 180,E1 -2207.597,E2 -2207.597} C_VEL
LIN {X 0,Y 573.228,Z 127.081,A -85,B 0,C 180,E1 -2210.392,E2 -2210.392} C_VEL
LIN {X 0,Y 573.229,Z 127.078,A -85,B 0,C 180,E1 -2213.076,E2 -2213.076} C_VEL
LIN {X 0,Y 573.247,Z 127.074,A -85,B 0,C 180,E1 -2215.67,E2 -2215.67} C_VEL
LIN {X 0,Y 573.226,Z 127.082,A -85,B 0,C 180,E1 -2218.184,E2 -2218.184} C_VEL
LIN {X 0,Y 573.239,Z 127.08,A -85,B 0,C 180,E1 -2220.633,E2 -2220.633} C_VEL
LIN {X 0,Y 573.212,Z 127.08,A -85,B 0,C 180,E1 -2223.513,E2 -2223.513} C_VEL
LIN {X 0,Y 573.222,Z 127.086,A -85,B 0,C 180,E1 -2226.512,E2 -2226.512} C_VEL
LIN {X 0,Y 573.269,Z 127.406,A -85,B 0,C 180,E1 -2226.609,E2 -2226.609} C_VEL
LIN {X 0,Y 573.959,Z 132.09,A -85,B 0,C 180,E1 -2227.312,E2 -2227.312} C_VEL
LIN {X 0,Y 573.824,Z 150.523,A -85,B 0,C 180,E1 -2229.944,E2 -2229.944} C_VEL
LIN {X 0,Y 573.588,Z 172.296,A -85,B 0,C 180,E1 -2233.015,E2 -2233.015} C_VEL
LIN {X 0,Y 573.407,Z 193.479,A -85,B 0,C 180,E1 -2235.991,E2 -2235.991} C_VEL
LIN {X 0,Y 573.389,Z 194.612,A -85,B 0,C 180,E1 -2236.149,E2 -2236.149} C_VEL
LIN {X 0,Y 574.049,Z 200.495,A -85,B 0,C 180,E1 -2236.256,E2 -2236.256} C_VEL
LIN {X 0,Y 573.883,Z 302.937,A -85,B 0,C 180,E1 -2237.557,E2 -2237.557} C_VEL
LIN {X 0,Y 573.779,Z 316.211,A -85,B 0,C 180,E1 -2237.869,E2 -2237.869} C_VEL
LIN {X 0,Y 573.699,Z 328.372,A -85,B 0,C 180,E1 -2238.294,E2 -2238.294} C_VEL
LIN {X 0,Y 573.586,Z 340.666,A -85,B 0,C 180,E1 -2238.876,E2 -2238.876} C_VEL
LIN {X 0,Y 573.428,Z 352.195,A -85,B 0,C 180,E1 -2239.585,E2 -2239.585} C_VEL
LIN {X 0,Y 573.333,Z 362.6,A -85,B 0,C 180,E1 -2240.385,E2 -2240.385} C_VEL
LIN {X 0,Y 573.241,Z 371.11,A -85,B 0,C 180,E1 -2241.184,E2 -2241.184} C_VEL
LIN {X 0,Y 573.161,Z 378.958,A -85,B 0,C 180,E1 -2242.071,E2 -2242.071} C_VEL
LIN {X 0,Y 573.073,Z 386.953,A -85,B 0,C 180,E1 -2243.185,E2 -2243.185} C_VEL
LIN {X 0,Y 573.07,Z 393.678,A -85,B 0,C 180,E1 -2244.369,E2 -2244.369} C_VEL
LIN {X 0,Y 573.028,Z 398.371,A -85,B 0,C 180,E1 -2245.427,E2 -2245.427} C_VEL
LIN {X 0,Y 573.022,Z 401.957,A -85,B 0,C 180,E1 -2246.484,E2 -2246.484} C_VEL
LIN {X 0,Y 572.959,Z 403.807,A -85,B 0,C 180,E1 -2247.187,E2 -2247.187} C_VEL
LIN {X 0,Y 572.946,Z 406.184,A -85,B 0,C 180,E1 -2248.594,E2 -2248.594} C_VEL
LIN {X 0,Y 572.938,Z 407,A -85,B 0,C 180,E1 -2250,E2 -2250} C_VEL
LIN {X 0,Y 572.946,Z 406.186,A -85,B 0,C 180,E1 -2251.405,E2 -2251.405} C_VEL
LIN {X 0,Y 572.94,Z 405.199,A -85,B 0,C 180,E1 -2252.109,E2 -2252.109} C_VEL
LIN {X 0,Y 572.959,Z 403.811,A -85,B 0,C 180,E1 -2252.812,E2 -2252.812} C_VEL
LIN {X 0,Y 573.014,Z 400.897,A -85,B 0,C 180,E1 -2253.868,E2 -2253.868} C_VEL
LIN {X 0,Y 572.963,Z 396.95,A -85,B 0,C 180,E1 -2254.925,E2 -2254.925} C_VEL
